Yaskawa INFORM job: DEMO_ROOF_SIDE_0625_3PAINT_43.JBI

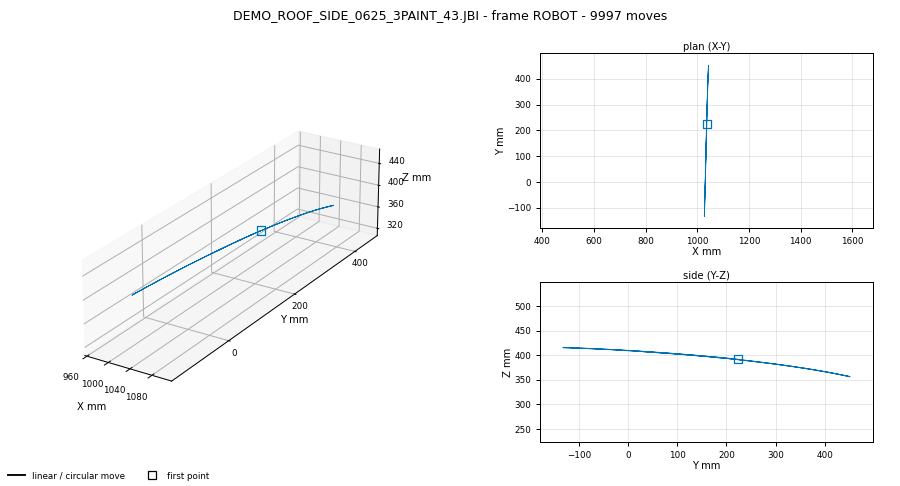
[picture p0: tool path of DEMO_ROOF_SIDE_0625_3PAINT_43.JBI in frame ROBOT, 9997 of 9997 moves have a stored position in this frame; points joined in program order, loops and branches not executed]
/JOB
//NAME DEMO_ROOF_SIDE_0625_3PAINT43
//POS
///NPOS 9997,0,0,0,0,0
///TOOL 0
///USER 0
///POSTYPE ROBOT
///RECTAN
///RCONF 1,0,0,0,0,0,0,0,0,0,0,0,0,0,0,0,0,0,0,0,0,0,0,0
C00000=1036.877,223.330,392.061,170.729,42.269,158.043
C00001=1036.870,223.081,392.088,170.727,42.268,158.043
C00002=1036.863,222.832,392.115,170.723,42.267,158.042
C00003=1036.857,222.584,392.143,170.721,42.266,158.042
C00004=1036.850,222.336,392.170,170.718,42.265,158.042
C00005=1036.844,222.088,392.198,170.716,42.264,158.041
C00006=1036.837,221.839,392.225,170.713,42.263,158.041
C00007=1036.830,221.591,392.252,170.711,42.262,158.040
C00008=1036.823,221.342,392.280,170.709,42.261,158.040
C00009=1036.817,221.094,392.307,170.705,42.261,158.040
C00010=1036.808,220.760,392.343,170.703,42.259,158.039
C00011=1036.799,220.427,392.380,170.699,42.258,158.039
C00012=1036.790,220.094,392.416,170.696,42.257,158.038
C00013=1036.782,219.761,392.454,170.692,42.255,158.038
C00014=1036.775,219.512,392.480,170.690,42.254,158.037
C00015=1036.768,219.264,392.508,170.687,42.254,158.037
C00016=1036.761,219.015,392.535,170.685,42.253,158.037
C00017=1036.754,218.767,392.562,170.683,42.252,158.036
C00018=1036.748,218.518,392.590,170.679,42.251,158.036
C00019=1036.741,218.270,392.616,170.677,42.251,158.036
C00020=1036.734,218.022,392.643,170.674,42.250,158.035
C00021=1036.727,217.773,392.670,170.672,42.249,158.035
C00022=1036.721,217.525,392.697,170.669,42.248,158.035
C00023=1036.714,217.276,392.724,170.667,42.247,158.034
C00024=1036.707,217.028,392.751,170.665,42.246,158.034
C00025=1036.701,216.779,392.778,170.662,42.245,158.034
C00026=1036.694,216.531,392.805,170.659,42.245,158.033
C00027=1036.687,216.282,392.832,170.657,42.244,158.033
C00028=1036.680,216.034,392.859,170.654,42.243,158.033
C00029=1036.674,215.785,392.886,170.652,42.242,158.032
C00030=1036.667,215.537,392.913,170.649,42.241,158.032
C00031=1036.660,215.288,392.940,170.647,42.240,158.031
C00032=1036.654,215.040,392.966,170.645,42.239,158.031
C00033=1036.647,214.792,392.994,170.642,42.238,158.031
C00034=1036.640,214.543,393.021,170.640,42.237,158.030
C00035=1036.634,214.295,393.048,170.637,42.236,158.030
C00036=1036.627,214.046,393.074,170.635,42.235,158.030
C00037=1036.620,213.797,393.101,170.633,42.234,158.029
C00038=1036.613,213.549,393.128,170.630,42.234,158.029
C00039=1036.607,213.301,393.155,170.628,42.233,158.029
C00040=1036.600,213.052,393.183,170.626,42.232,158.028
C00041=1036.593,212.804,393.209,170.622,42.231,158.028
C00042=1036.588,212.555,393.236,170.620,42.230,158.028
C00043=1036.580,212.307,393.263,170.617,42.229,158.027
C00044=1036.574,212.058,393.290,170.615,42.228,158.027
C00045=1036.567,211.810,393.316,170.612,42.227,158.027
C00046=1036.561,211.561,393.343,170.610,42.226,158.026
C00047=1036.553,211.313,393.370,170.608,42.226,158.026
C00048=1036.547,211.065,393.396,170.605,42.225,158.025
C00049=1036.541,210.816,393.423,170.603,42.224,158.025
C00050=1036.533,210.567,393.450,170.601,42.223,158.025
C00051=1036.527,210.319,393.477,170.598,42.222,158.025
C00052=1036.520,210.070,393.504,170.596,42.221,158.024
C00053=1036.513,209.822,393.530,170.593,42.220,158.024
C00054=1036.507,209.573,393.557,170.591,42.219,158.023
C00055=1036.500,209.325,393.583,170.589,42.219,158.023
C00056=1036.493,209.077,393.610,170.586,42.218,158.023
C00057=1036.487,208.828,393.637,170.584,42.217,158.022
C00058=1036.480,208.579,393.663,170.582,42.216,158.022
C00059=1036.473,208.331,393.689,170.579,42.215,158.022
C00060=1036.466,208.083,393.716,170.577,42.214,158.021
C00061=1036.460,207.834,393.743,170.574,42.213,158.021
C00062=1036.453,207.585,393.769,170.572,42.213,158.021
C00063=1036.446,207.337,393.795,170.570,42.212,158.020
C00064=1036.440,207.089,393.821,170.567,42.211,158.020
C00065=1036.433,206.840,393.848,170.565,42.210,158.020
C00066=1036.424,206.513,393.883,170.561,42.209,158.019
C00067=1036.415,206.185,393.919,170.559,42.208,158.019
C00068=1036.406,205.857,393.953,170.555,42.207,158.019
C00069=1036.398,205.530,393.988,170.552,42.206,158.018
C00070=1036.371,204.480,394.094,170.239,42.102,157.976
C00071=1036.365,204.230,394.118,170.236,42.101,157.976
C00072=1036.359,203.982,394.144,170.233,42.101,157.976
C00073=1036.353,203.733,394.169,170.230,42.101,157.975
C00074=1036.347,203.484,394.194,170.226,42.101,157.975
C00075=1036.340,203.236,394.220,170.223,42.101,157.975
C00076=1036.335,202.987,394.244,170.220,42.100,157.975
C00077=1036.329,202.739,394.269,170.217,42.100,157.974
C00078=1036.322,202.490,394.294,170.214,42.101,157.974
C00079=1036.316,202.241,394.319,170.211,42.100,157.974
C00080=1036.310,201.992,394.344,170.206,42.100,157.974
C00081=1036.304,201.744,394.369,170.203,42.100,157.973
C00082=1036.298,201.496,394.394,170.200,42.100,157.973
C00083=1036.292,201.246,394.419,170.197,42.100,157.973
C00084=1036.286,200.998,394.444,170.194,42.100,157.973
C00085=1036.280,200.749,394.470,170.190,42.100,157.973
C00086=1036.273,200.500,394.494,170.187,42.100,157.972
C00087=1036.267,200.251,394.519,170.184,42.100,157.972
C00088=1036.261,200.003,394.543,170.181,42.100,157.972
C00089=1036.255,199.754,394.568,170.178,42.100,157.972
C00090=1036.248,199.505,394.592,170.174,42.100,157.972
C00091=1036.242,199.257,394.617,170.171,42.100,157.971
C00092=1036.236,199.008,394.643,170.168,42.100,157.971
C00093=1036.230,198.760,394.666,170.165,42.100,157.971
C00094=1036.224,198.510,394.691,170.162,42.100,157.971
C00095=1036.217,198.262,394.716,170.159,42.100,157.971
C00096=1036.211,198.013,394.740,170.156,42.101,157.970
C00097=1036.204,197.764,394.765,170.152,42.100,157.970
C00098=1036.199,197.516,394.789,170.149,42.100,157.970
C00099=1036.192,197.268,394.814,170.146,42.101,157.970
C00100=1036.186,197.018,394.839,170.142,42.101,157.970
C00101=1036.179,196.770,394.863,170.139,42.100,157.969
C00102=1036.173,196.521,394.888,170.136,42.101,157.969
C00103=1036.167,196.272,394.912,170.132,42.101,157.969
C00104=1036.161,196.024,394.937,170.129,42.101,157.969
C00105=1036.155,195.774,394.962,170.126,42.101,157.969
C00106=1036.149,195.526,394.985,170.123,42.101,157.968
C00107=1036.142,195.277,395.011,170.120,42.101,157.968
C00108=1036.136,195.028,395.035,170.117,42.101,157.968
C00109=1036.131,194.780,395.059,170.114,42.101,157.968
C00110=1036.124,194.531,395.084,170.110,42.101,157.968
C00111=1036.118,194.282,395.108,170.107,42.102,157.968
C00112=1036.112,194.034,395.132,170.104,42.102,157.967
C00113=1036.105,193.785,395.157,170.101,42.101,157.967
C00114=1036.099,193.536,395.181,170.099,42.102,157.967
C00115=1036.093,193.288,395.206,170.096,42.101,157.967
C00116=1036.087,193.039,395.230,170.093,42.102,157.967
C00117=1036.081,192.790,395.255,170.089,42.102,157.966
C00118=1036.075,192.542,395.279,170.086,42.102,157.966
C00119=1036.069,192.292,395.303,170.083,42.102,157.966
C00120=1036.063,192.044,395.327,170.080,42.102,157.966
C00121=1036.057,191.795,395.352,170.077,42.102,157.966
C00122=1036.050,191.547,395.376,170.074,42.102,157.965
C00123=1036.045,191.298,395.401,170.071,42.102,157.965
C00124=1036.038,191.049,395.425,170.067,42.102,157.965
C00125=1036.033,190.800,395.449,170.064,42.103,157.965
C00126=1036.026,190.551,395.473,170.061,42.103,157.965
C00127=1036.020,190.302,395.497,170.058,42.103,157.965
C00128=1036.014,190.054,395.522,170.055,42.103,157.964
C00129=1036.008,189.805,395.546,170.052,42.103,157.964
C00130=1036.002,189.557,395.570,170.049,42.103,157.964
C00131=1035.995,189.272,395.597,170.046,42.103,157.964
C00132=1035.988,188.989,395.625,170.042,42.103,157.964
C00133=1035.981,188.704,395.653,170.038,42.104,157.964
C00134=1035.974,188.420,395.680,170.035,42.104,157.963
C00135=1035.968,188.171,395.705,170.032,42.103,157.963
C00136=1035.962,187.923,395.729,170.029,42.104,157.963
C00137=1035.956,187.673,395.753,170.026,42.104,157.963
C00138=1035.950,187.425,395.777,170.024,42.104,157.963
C00139=1035.944,187.176,395.801,170.020,42.104,157.962
C00140=1035.938,186.927,395.825,170.017,42.104,157.962
C00141=1035.932,186.678,395.850,170.014,42.105,157.962
C00142=1035.926,186.430,395.873,170.011,42.105,157.962
C00143=1035.921,186.181,395.898,170.008,42.105,157.962
C00144=1035.914,185.932,395.922,170.005,42.105,157.962
C00145=1035.909,185.684,395.946,170.002,42.105,157.961
C00146=1035.903,185.435,395.970,170.000,42.105,157.961
C00147=1035.896,185.186,395.994,169.997,42.105,157.961
C00148=1035.891,184.937,396.018,169.993,42.105,157.961
C00149=1035.885,184.689,396.042,169.990,42.106,157.961
C00150=1035.879,184.440,396.067,169.987,42.105,157.961
C00151=1035.873,184.191,396.090,169.984,42.106,157.960
C00152=1035.867,183.943,396.114,169.982,42.105,157.960
C00153=1035.861,183.693,396.138,169.979,42.106,157.960
C00154=1035.856,183.445,396.162,169.976,42.106,157.960
C00155=1035.849,183.196,396.186,169.972,42.106,157.960
C00156=1035.843,182.947,396.210,169.969,42.107,157.960
C00157=1035.837,182.698,396.233,169.966,42.107,157.960
C00158=1035.831,182.449,396.257,169.963,42.108,157.959
C00159=1035.823,182.201,396.280,169.960,42.108,157.959
C00160=1035.818,181.952,396.303,169.957,42.108,157.959
C00161=1035.811,181.703,396.327,169.955,42.108,157.959
C00162=1035.805,181.454,396.350,169.952,42.109,157.959
C00163=1035.799,181.205,396.374,169.949,42.109,157.959
C00164=1035.793,180.957,396.398,169.946,42.109,157.959
C00165=1035.787,180.708,396.421,169.943,42.110,157.959
C00166=1035.780,180.459,396.445,169.940,42.110,157.958
C00167=1035.774,180.210,396.468,169.937,42.110,157.958
C00168=1035.767,179.961,396.491,169.934,42.111,157.958
C00169=1035.761,179.712,396.514,169.931,42.111,157.958
C00170=1035.755,179.463,396.538,169.929,42.111,157.958
C00171=1035.749,179.215,396.562,169.926,42.112,157.958
C00172=1035.743,178.966,396.585,169.923,42.112,157.958
C00173=1035.736,178.717,396.609,169.919,42.113,157.958
C00174=1035.731,178.468,396.632,169.916,42.113,157.958
C00175=1035.723,178.220,396.655,169.913,42.114,157.957
C00176=1035.717,177.971,396.678,169.910,42.113,157.957
C00177=1035.712,177.722,396.701,169.908,42.114,157.957
C00178=1035.705,177.473,396.725,169.905,42.114,157.957
C00179=1035.699,177.224,396.748,169.902,42.115,157.957
C00180=1035.693,176.975,396.772,169.899,42.115,157.957
C00181=1035.687,176.726,396.795,169.896,42.115,157.957
C00182=1035.680,176.478,396.818,169.893,42.116,157.957
C00183=1035.674,176.229,396.841,169.891,42.116,157.957
C00184=1035.668,175.980,396.864,169.888,42.117,157.956
C00185=1035.662,175.731,396.888,169.885,42.117,157.956
C00186=1035.656,175.482,396.911,169.882,42.117,157.956
C00187=1035.650,175.234,396.935,169.879,42.117,157.956
C00188=1035.644,174.985,396.958,169.876,42.118,157.956
C00189=1035.637,174.736,396.980,169.874,42.118,157.956
C00190=1035.631,174.487,397.004,169.871,42.118,157.956
C00191=1035.625,174.238,397.027,169.867,42.119,157.956
C00192=1035.619,173.989,397.050,169.864,42.119,157.955
C00193=1035.613,173.740,397.074,169.861,42.120,157.955
C00194=1035.607,173.491,397.097,169.859,42.120,157.955
C00195=1035.600,173.207,397.123,169.855,42.121,157.955
C00196=1035.592,172.922,397.149,169.852,42.121,157.955
C00197=1035.586,172.638,397.176,169.849,42.122,157.955
C00198=1035.579,172.354,397.202,169.846,42.122,157.955
C00199=1035.573,172.104,397.225,169.843,42.122,157.955
C00200=1035.567,171.856,397.249,169.840,42.122,157.954
C00201=1035.561,171.607,397.272,169.838,42.123,157.954
C00202=1035.554,171.359,397.294,169.835,42.123,157.954
C00203=1035.548,171.109,397.318,169.832,42.123,157.954
C00204=1035.542,170.860,397.341,169.829,42.124,157.954
C00205=1035.536,170.612,397.364,169.827,42.124,157.954
C00206=1035.531,170.363,397.387,169.824,42.125,157.954
C00207=1035.525,170.114,397.410,169.821,42.125,157.954
C00208=1035.518,169.865,397.433,169.818,42.126,157.954
C00209=1035.512,169.616,397.456,169.816,42.126,157.954
C00210=1035.506,169.367,397.479,169.813,42.126,157.953
C00211=1035.500,169.119,397.503,169.810,42.127,157.953
C00212=1035.495,168.870,397.525,169.807,42.127,157.953
C00213=1035.488,168.621,397.548,169.804,42.127,157.953
C00214=1035.482,168.371,397.571,169.801,42.128,157.953
C00215=1035.476,168.123,397.594,169.798,42.128,157.953
C00216=1035.470,167.874,397.617,169.796,42.129,157.953
C00217=1035.465,167.625,397.640,169.793,42.129,157.953
C00218=1035.458,167.376,397.662,169.790,42.129,157.953
C00219=1035.452,167.127,397.685,169.787,42.129,157.952
C00220=1035.447,166.878,397.708,169.785,42.130,157.952
C00221=1035.441,166.630,397.732,169.782,42.130,157.952
C00222=1035.434,166.381,397.755,169.779,42.131,157.952
C00223=1035.428,166.132,397.778,169.777,42.131,157.952
C00224=1035.422,165.883,397.800,169.774,42.131,157.952
C00225=1035.416,165.634,397.823,169.771,42.132,157.952
C00226=1035.411,165.385,397.846,169.769,42.132,157.952
C00227=1035.404,165.137,397.869,169.766,42.132,157.952
C00228=1035.398,164.888,397.892,169.763,42.133,157.952
C00229=1035.393,164.639,397.915,169.761,42.133,157.951
C00230=1035.387,164.390,397.938,169.758,42.134,157.951
C00231=1035.381,164.141,397.960,169.755,42.134,157.951
C00232=1035.375,163.893,397.983,169.753,42.134,157.951
C00233=1035.369,163.643,398.005,169.750,42.135,157.951
C00234=1035.364,163.394,398.028,169.747,42.135,157.951
C00235=1035.358,163.145,398.051,169.745,42.136,157.951
C00236=1035.351,162.897,398.073,169.742,42.136,157.951
C00237=1035.346,162.648,398.096,169.738,42.136,157.951
C00238=1035.340,162.399,398.119,169.736,42.137,157.951
C00239=1035.334,162.150,398.142,169.733,42.137,157.951
C00240=1035.328,161.901,398.164,169.730,42.138,157.950
C00241=1035.322,161.652,398.187,169.728,42.138,157.950
C00242=1035.316,161.404,398.210,169.725,42.138,157.950
C00243=1035.311,161.154,398.233,169.722,42.139,157.950
C00244=1035.304,160.905,398.255,169.720,42.139,157.950
C00245=1035.299,160.657,398.278,169.717,42.140,157.950
C00246=1035.293,160.408,398.301,169.715,42.140,157.950
C00247=1035.287,160.159,398.324,169.712,42.140,157.950
C00248=1035.282,159.909,398.346,169.709,42.141,157.950
C00249=1035.275,159.661,398.368,169.707,42.141,157.950
C00250=1035.269,159.412,398.391,169.704,42.141,157.949
C00251=1035.263,159.163,398.414,169.701,42.142,157.949
C00252=1035.257,158.914,398.435,169.699,42.142,157.949
C00253=1035.250,158.665,398.458,169.696,42.143,157.949
C00254=1035.245,158.416,398.480,169.693,42.144,157.949
C00255=1035.238,158.167,398.503,169.691,42.144,157.949
C00256=1035.232,157.918,398.525,169.688,42.145,157.949
C00257=1035.226,157.668,398.547,169.685,42.145,157.949
C00258=1035.220,157.421,398.569,169.683,42.146,157.949
C00259=1035.213,157.135,398.595,169.679,42.146,157.949
C00260=1035.206,156.850,398.620,169.676,42.147,157.949
C00261=1035.199,156.565,398.646,169.673,42.147,157.949
C00262=1035.192,156.280,398.671,169.670,42.148,157.949
C00263=1035.186,156.032,398.694,169.668,42.149,157.949
C00264=1035.180,155.782,398.716,169.665,42.149,157.948
C00265=1035.174,155.533,398.738,169.662,42.150,157.948
C00266=1035.168,155.284,398.760,169.660,42.150,157.948
C00267=1035.162,155.035,398.783,169.657,42.151,157.948
C00268=1035.156,154.786,398.804,169.655,42.151,157.948
C00269=1035.150,154.538,398.826,169.652,42.152,157.948
C00270=1035.144,154.289,398.848,169.649,42.152,157.948
C00271=1035.138,154.040,398.871,169.647,42.153,157.948
C00272=1035.132,153.791,398.893,169.644,42.154,157.948
C00273=1035.125,153.542,398.915,169.641,42.154,157.948
C00274=1035.119,153.293,398.937,169.639,42.154,157.948
C00275=1035.114,153.044,398.959,169.636,42.155,157.948
C00276=1035.107,152.795,398.981,169.633,42.156,157.948
C00277=1035.101,152.546,399.003,169.631,42.156,157.948
C00278=1035.095,152.297,399.025,169.628,42.157,157.948
C00279=1035.088,152.048,399.047,169.626,42.158,157.948
C00280=1035.082,151.799,399.068,169.623,42.158,157.947
C00281=1035.077,151.551,399.091,169.620,42.158,157.947
C00282=1035.071,151.301,399.113,169.618,42.159,157.947
C00283=1035.065,151.052,399.134,169.615,42.160,157.947
C00284=1035.058,150.804,399.157,169.613,42.160,157.947
C00285=1035.052,150.554,399.178,169.610,42.161,157.947
C00286=1035.046,150.305,399.200,169.607,42.162,157.947
C00287=1035.040,150.056,399.223,169.605,42.162,157.947
C00288=1035.034,149.807,399.244,169.602,42.162,157.947
C00289=1035.029,149.559,399.266,169.601,42.163,157.947
C00290=1035.022,149.310,399.288,169.598,42.164,157.947
C00291=1035.016,149.061,399.310,169.594,42.164,157.947
C00292=1035.010,148.812,399.331,169.593,42.165,157.947
C00293=1035.004,148.562,399.353,169.590,42.166,157.947
C00294=1034.998,148.314,399.376,169.588,42.166,157.947
C00295=1034.992,148.065,399.397,169.585,42.166,157.947
C00296=1034.986,147.816,399.419,169.582,42.167,157.947
C00297=1034.980,147.567,399.440,169.580,42.168,157.947
C00298=1034.974,147.318,399.463,169.577,42.168,157.946
C00299=1034.967,147.069,399.484,169.575,42.169,157.947
C00300=1034.961,146.820,399.506,169.572,42.170,157.946
C00301=1034.956,146.571,399.527,169.569,42.171,157.946
C00302=1034.949,146.322,399.549,169.567,42.171,157.946
C00303=1034.943,146.073,399.571,169.564,42.171,157.946
C00304=1034.937,145.823,399.592,169.562,42.172,157.946
C00305=1034.931,145.574,399.614,169.559,42.173,157.946
C00306=1034.925,145.326,399.636,169.556,42.174,157.946
C00307=1034.918,145.078,399.657,169.554,42.174,157.946
C00308=1034.912,144.828,399.679,169.551,42.175,157.946
C00309=1034.906,144.579,399.700,169.549,42.176,157.946
C00310=1034.900,144.330,399.722,169.546,42.176,157.946
C00311=1034.894,144.081,399.743,169.544,42.177,157.946
C00312=1034.888,143.832,399.765,169.541,42.177,157.946
C00313=1034.882,143.583,399.786,169.538,42.178,157.946
C00314=1034.876,143.334,399.808,169.536,42.179,157.946
C00315=1034.870,143.085,399.830,169.533,42.179,157.946
C00316=1034.864,142.836,399.851,169.532,42.180,157.946
C00317=1034.857,142.587,399.872,169.528,42.181,157.946
C00318=1034.851,142.338,399.894,169.527,42.182,157.946
C00319=1034.845,142.089,399.915,169.524,42.182,157.946
C00320=1034.839,141.840,399.936,169.521,42.183,157.946
C00321=1034.833,141.591,399.958,169.519,42.183,157.946
C00322=1034.827,141.342,399.980,169.516,42.184,157.946
C00323=1034.821,141.056,400.004,169.513,42.185,157.946
C00324=1034.813,140.771,400.028,169.511,42.185,157.946
C00325=1034.807,140.486,400.053,169.508,42.186,157.946
C00326=1034.799,140.200,400.077,169.505,42.187,157.945
C00327=1034.794,139.952,400.099,169.502,42.187,157.945
C00328=1034.787,139.702,400.120,169.500,42.188,157.945
C00329=1034.781,139.453,400.142,169.497,42.189,157.945
C00330=1034.776,139.205,400.163,169.495,42.190,157.945
C00331=1034.769,138.956,400.184,169.492,42.190,157.945
C00332=1034.763,138.707,400.206,169.490,42.191,157.945
C00333=1034.756,138.457,400.227,169.487,42.191,157.945
C00334=1034.751,138.208,400.248,169.484,42.193,157.945
C00335=1034.744,137.959,400.269,169.482,42.193,157.945
C00336=1034.738,137.710,400.291,169.479,42.193,157.945
C00337=1034.733,137.462,400.312,169.477,42.194,157.945
C00338=1034.726,137.213,400.333,169.474,42.195,157.945
C00339=1034.720,136.963,400.354,169.473,42.196,157.945
C00340=1034.714,136.715,400.375,169.470,42.196,157.945
C00341=1034.708,136.465,400.397,169.468,42.197,157.945
C00342=1034.701,136.216,400.418,169.465,42.197,157.945
C00343=1034.696,135.967,400.438,169.463,42.198,157.945
C00344=1034.690,135.718,400.460,169.460,42.199,157.945
C00345=1034.683,135.469,400.481,169.458,42.200,157.945
C00346=1034.678,135.220,400.502,169.455,42.201,157.945
C00347=1034.671,134.971,400.523,169.452,42.201,157.945
C00348=1034.664,134.722,400.544,169.450,42.202,157.945
C00349=1034.659,134.473,400.565,169.447,42.203,157.945
C00350=1034.652,134.224,400.586,169.445,42.204,157.945
C00351=1034.647,133.975,400.607,169.442,42.204,157.945
C00352=1034.641,133.726,400.628,169.440,42.205,157.945
C00353=1034.634,133.477,400.649,169.437,42.206,157.945
C00354=1034.628,133.228,400.670,169.436,42.206,157.945
C00355=1034.622,132.979,400.691,169.433,42.207,157.945
C00356=1034.616,132.730,400.712,169.431,42.208,157.945
C00357=1034.610,132.481,400.734,169.428,42.208,157.945
C00358=1034.604,132.231,400.754,169.426,42.209,157.945
C00359=1034.598,131.983,400.775,169.423,42.210,157.945
C00360=1034.592,131.733,400.796,169.421,42.211,157.945
C00361=1034.586,131.485,400.817,169.418,42.211,157.944
C00362=1034.580,131.235,400.838,169.416,42.212,157.945
C00363=1034.573,130.986,400.859,169.413,42.212,157.944
C00364=1034.568,130.737,400.879,169.411,42.213,157.945
C00365=1034.561,130.488,400.900,169.408,42.214,157.944
C00366=1034.556,130.239,400.921,169.406,42.215,157.944
C00367=1034.549,129.990,400.942,169.403,42.216,157.944
C00368=1034.542,129.741,400.962,169.401,42.216,157.944
C00369=1034.537,129.492,400.984,169.399,42.217,157.944
C00370=1034.530,129.243,401.004,169.397,42.218,157.945
C00371=1034.524,128.994,401.025,169.394,42.219,157.944
C00372=1034.517,128.745,401.045,169.392,42.220,157.944
C00373=1034.511,128.495,401.066,169.389,42.221,157.944
C00374=1034.505,128.247,401.087,169.387,42.221,157.944
C00375=1034.498,127.997,401.107,169.384,42.222,157.944
C00376=1034.493,127.748,401.127,169.382,42.223,157.944
C00377=1034.486,127.499,401.148,169.379,42.224,157.944
C00378=1034.480,127.251,401.168,169.376,42.225,157.944
C00379=1034.474,127.001,401.190,169.375,42.226,157.944
C00380=1034.468,126.753,401.210,169.371,42.226,157.944
C00381=1034.461,126.503,401.230,169.370,42.227,157.944
C00382=1034.455,126.254,401.251,169.367,42.228,157.944
C00383=1034.449,126.005,401.272,169.365,42.228,157.944
C00384=1034.443,125.756,401.292,169.362,42.229,157.944
C00385=1034.437,125.507,401.312,169.360,42.230,157.944
C00386=1034.431,125.258,401.334,169.357,42.231,157.944
C00387=1034.423,124.972,401.357,169.355,42.232,157.944
C00388=1034.416,124.687,401.381,169.352,42.233,157.944
C00389=1034.409,124.401,401.403,169.350,42.234,157.944
C00390=1034.402,124.116,401.427,169.346,42.234,157.944
C00391=1034.396,123.867,401.448,169.345,42.235,157.944
C00392=1034.390,123.618,401.469,169.342,42.237,157.944
C00393=1034.384,123.369,401.489,169.340,42.237,157.944
C00394=1034.377,123.119,401.509,169.337,42.238,157.944
C00395=1034.371,122.870,401.529,169.335,42.238,157.944
C00396=1034.365,122.621,401.551,169.332,42.239,157.944
C00397=1034.359,122.372,401.571,169.330,42.240,157.944
C00398=1034.353,122.124,401.591,169.327,42.241,157.944
C00399=1034.347,121.874,401.611,169.325,42.242,157.944
C00400=1034.341,121.625,401.631,169.322,42.243,157.944
C00401=1034.334,121.376,401.652,169.320,42.243,157.944
C00402=1034.328,121.127,401.672,169.318,42.244,157.944
C00403=1034.323,120.877,401.693,169.316,42.245,157.944
C00404=1034.317,120.629,401.713,169.314,42.245,157.944
C00405=1034.311,120.380,401.733,169.311,42.246,157.944
C00406=1034.304,120.130,401.754,169.309,42.247,157.944
C00407=1034.298,119.882,401.775,169.306,42.248,157.944
C00408=1034.292,119.632,401.795,169.304,42.249,157.944
C00409=1034.286,119.384,401.815,169.301,42.249,157.944
C00410=1034.280,119.135,401.835,169.299,42.250,157.944
C00411=1034.274,118.885,401.856,169.296,42.251,157.944
C00412=1034.268,118.636,401.876,169.294,42.252,157.944
C00413=1034.261,118.387,401.896,169.293,42.253,157.944
C00414=1034.255,118.138,401.916,169.289,42.253,157.944
C00415=1034.250,117.889,401.937,169.288,42.254,157.944
C00416=1034.244,117.639,401.957,169.285,42.255,157.944
C00417=1034.237,117.391,401.978,169.283,42.255,157.944
C00418=1034.231,117.142,401.998,169.280,42.256,157.944
C00419=1034.225,116.892,402.019,169.278,42.257,157.944
C00420=1034.219,116.643,402.039,169.276,42.258,157.944
C00421=1034.213,116.395,402.059,169.273,42.259,157.944
C00422=1034.207,116.145,402.079,169.271,42.259,157.944
C00423=1034.202,115.896,402.099,169.268,42.260,157.944
C00424=1034.196,115.647,402.119,169.266,42.261,157.944
C00425=1034.189,115.398,402.140,169.263,42.262,157.944
C00426=1034.183,115.149,402.160,169.261,42.262,157.944
C00427=1034.177,114.900,402.180,169.260,42.263,157.944
C00428=1034.171,114.650,402.201,169.257,42.264,157.944
C00429=1034.165,114.401,402.221,169.255,42.264,157.944
C00430=1034.159,114.153,402.241,169.252,42.265,157.944
C00431=1034.153,113.903,402.261,169.250,42.266,157.944
C00432=1034.148,113.653,402.281,169.248,42.267,157.944
C00433=1034.142,113.405,402.301,169.245,42.268,157.944
C00434=1034.135,113.155,402.321,169.243,42.268,157.944
C00435=1034.129,112.906,402.341,169.240,42.269,157.944
C00436=1034.123,112.657,402.361,169.238,42.270,157.944
C00437=1034.116,112.408,402.381,169.236,42.270,157.944
C00438=1034.110,112.159,402.401,169.233,42.271,157.944
C00439=1034.105,111.910,402.420,169.232,42.272,157.944
C00440=1034.099,111.661,402.440,169.229,42.274,157.944
C00441=1034.092,111.411,402.461,169.227,42.274,157.944
C00442=1034.086,111.162,402.481,169.224,42.275,157.944
C00443=1034.080,110.914,402.501,169.222,42.276,157.944
C00444=1034.074,110.664,402.520,169.220,42.276,157.944
C00445=1034.068,110.415,402.540,169.217,42.277,157.944
C00446=1034.061,110.166,402.560,169.215,42.278,157.944
C00447=1034.055,109.917,402.580,169.213,42.279,157.944
C00448=1034.049,109.667,402.599,169.210,42.280,157.944
C00449=1034.043,109.418,402.619,169.208,42.281,157.944
C00450=1034.037,109.170,402.639,169.206,42.282,157.944
C00451=1034.029,108.884,402.661,169.203,42.283,157.944
C00452=1034.022,108.598,402.684,169.200,42.284,157.944
C00453=1034.015,108.312,402.707,169.198,42.285,157.944
C00454=1034.008,108.027,402.729,169.195,42.286,157.944
C00455=1034.002,107.778,402.749,169.192,42.286,157.944
C00456=1033.996,107.529,402.769,169.190,42.287,157.944
C00457=1033.989,107.279,402.788,169.188,42.288,157.944
C00458=1033.983,107.030,402.808,169.186,42.289,157.944
C00459=1033.977,106.781,402.827,169.184,42.290,157.944
C00460=1033.971,106.532,402.847,169.181,42.291,157.944
C00461=1033.965,106.282,402.867,169.179,42.292,157.944
C00462=1033.958,106.033,402.886,169.176,42.293,157.944
C00463=1033.952,105.785,402.906,169.174,42.294,157.944
C00464=1033.946,105.536,402.926,169.171,42.294,157.944
C00465=1033.940,105.286,402.945,169.170,42.295,157.944
C00466=1033.933,105.037,402.965,169.168,42.296,157.944
C00467=1033.927,104.788,402.984,169.165,42.297,157.944
C00468=1033.921,104.539,403.004,169.163,42.298,157.944
C00469=1033.916,104.289,403.023,169.160,42.299,157.944
C00470=1033.910,104.041,403.043,169.158,42.300,157.944
C00471=1033.903,103.791,403.062,169.156,42.301,157.945
C00472=1033.897,103.542,403.082,169.153,42.301,157.944
C00473=1033.891,103.293,403.102,169.151,42.302,157.944
C00474=1033.885,103.044,403.122,169.149,42.303,157.945
C00475=1033.878,102.795,403.141,169.147,42.304,157.945
C00476=1033.873,102.546,403.160,169.145,42.304,157.944
C00477=1033.866,102.296,403.180,169.142,42.305,157.945
C00478=1033.860,102.047,403.200,169.140,42.306,157.945
C00479=1033.854,101.798,403.219,169.137,42.308,157.945
C00480=1033.848,101.549,403.238,169.135,42.308,157.945
C00481=1033.842,101.299,403.258,169.133,42.309,157.945
C00482=1033.836,101.051,403.278,169.130,42.310,157.945
C00483=1033.829,100.801,403.297,169.129,42.311,157.945
C00484=1033.823,100.552,403.316,169.127,42.311,157.945
C00485=1033.818,100.303,403.336,169.124,42.312,157.945
C00486=1033.812,100.054,403.356,169.122,42.313,157.945
C00487=1033.805,99.805,403.374,169.119,42.314,157.945
C00488=1033.799,99.555,403.394,169.117,42.315,157.945
C00489=1033.792,99.306,403.413,169.114,42.316,157.945
C00490=1033.786,99.057,403.433,169.112,42.317,157.945
C00491=1033.780,98.807,403.451,169.110,42.318,157.945
C00492=1033.774,98.559,403.471,169.108,42.319,157.945
C00493=1033.768,98.310,403.490,169.106,42.320,157.945
C00494=1033.762,98.060,403.509,169.103,42.321,157.945
C00495=1033.755,97.811,403.528,169.101,42.321,157.945
C00496=1033.749,97.562,403.548,169.099,42.322,157.945
C00497=1033.742,97.312,403.567,169.096,42.323,157.945
C00498=1033.737,97.063,403.586,169.094,42.324,157.945
C00499=1033.730,96.814,403.605,169.091,42.325,157.945
C00500=1033.724,96.565,403.625,169.090,42.326,157.945
C00501=1033.718,96.316,403.643,169.088,42.327,157.945
C00502=1033.712,96.066,403.662,169.085,42.328,157.945
C00503=1033.706,95.818,403.682,169.083,42.329,157.945
C00504=1033.699,95.569,403.700,169.080,42.330,157.945
C00505=1033.693,95.319,403.720,169.078,42.331,157.945
C00506=1033.687,95.070,403.738,169.076,42.332,157.945
C00507=1033.681,94.820,403.758,169.073,42.333,157.945
C00508=1033.674,94.572,403.777,169.071,42.333,157.945
C00509=1033.668,94.322,403.797,169.069,42.334,157.945
C00510=1033.662,94.073,403.815,169.067,42.335,157.945
C00511=1033.656,93.824,403.834,169.065,42.336,157.945
C00512=1033.650,93.574,403.853,169.062,42.337,157.945
C00513=1033.644,93.325,403.872,169.060,42.337,157.945
C00514=1033.637,93.077,403.892,169.057,42.338,157.945
C00515=1033.631,92.791,403.913,169.055,42.339,157.945
C00516=1033.623,92.505,403.935,169.053,42.341,157.945
C00517=1033.616,92.219,403.957,169.050,42.342,157.945
C00518=1033.609,91.934,403.979,169.047,42.343,157.945
C00519=1033.603,91.685,403.998,169.045,42.344,157.945
C00520=1033.597,91.435,404.017,169.043,42.345,157.945
C00521=1033.591,91.186,404.035,169.040,42.345,157.945
C00522=1033.585,90.937,404.055,169.038,42.346,157.945
C00523=1033.579,90.688,404.073,169.036,42.347,157.945
C00524=1033.573,90.438,404.093,169.034,42.348,157.945
C00525=1033.567,90.189,404.111,169.032,42.349,157.946
C00526=1033.561,89.940,404.130,169.029,42.350,157.945
C00527=1033.554,89.691,404.149,169.027,42.351,157.945
C00528=1033.548,89.441,404.168,169.025,42.351,157.946
C00529=1033.542,89.192,404.186,169.022,42.353,157.946
C00530=1033.535,88.943,404.205,169.020,42.354,157.946
C00531=1033.530,88.694,404.224,169.017,42.355,157.946
C00532=1033.523,88.445,404.243,169.016,42.356,157.946
C00533=1033.517,88.196,404.262,169.014,42.357,157.946
C00534=1033.510,87.946,404.280,169.011,42.358,157.946
C00535=1033.504,87.697,404.299,169.009,42.359,157.946
C00536=1033.497,87.448,404.318,169.006,42.360,157.946
C00537=1033.492,87.199,404.337,169.004,42.361,157.946
C00538=1033.485,86.950,404.355,169.002,42.361,157.946
C00539=1033.479,86.701,404.374,168.999,42.362,157.946
C00540=1033.472,86.451,404.393,168.998,42.363,157.946
C00541=1033.466,86.202,404.411,168.995,42.364,157.946
C00542=1033.460,85.953,404.429,168.993,42.365,157.946
C00543=1033.454,85.703,404.449,168.991,42.366,157.946
C00544=1033.448,85.454,404.467,168.988,42.367,157.946
C00545=1033.441,85.205,404.486,168.986,42.368,157.946
C00546=1033.435,84.956,404.505,168.984,42.369,157.946
C00547=1033.428,84.707,404.523,168.982,42.370,157.946
C00548=1033.422,84.457,404.541,168.980,42.371,157.946
C00549=1033.417,84.207,404.560,168.977,42.372,157.946
C00550=1033.410,83.958,404.579,168.975,42.373,157.946
C00551=1033.404,83.709,404.598,168.972,42.374,157.946
C00552=1033.398,83.461,404.616,168.970,42.375,157.946
C00553=1033.392,83.212,404.635,168.968,42.376,157.946
C00554=1033.385,82.962,404.653,168.966,42.377,157.946
C00555=1033.379,82.713,404.671,168.964,42.378,157.946
C00556=1033.373,82.463,404.690,168.961,42.379,157.946
C00557=1033.367,82.214,404.709,168.959,42.379,157.946
C00558=1033.361,81.964,404.727,168.957,42.380,157.946
C00559=1033.354,81.715,404.746,168.954,42.381,157.946
C00560=1033.348,81.466,404.764,168.952,42.382,157.946
C00561=1033.342,81.217,404.783,168.951,42.383,157.947
C00562=1033.336,80.968,404.800,168.948,42.384,157.947
C00563=1033.330,80.719,404.820,168.946,42.385,157.947
C00564=1033.324,80.470,404.838,168.943,42.386,157.947
C00565=1033.317,80.220,404.857,168.941,42.387,157.947
C00566=1033.311,79.971,404.875,168.939,42.388,157.947
C00567=1033.305,79.722,404.894,168.936,42.389,157.947
C00568=1033.298,79.472,404.912,168.934,42.390,157.947
C00569=1033.293,79.223,404.930,168.933,42.391,157.947
C00570=1033.287,78.974,404.949,168.930,42.392,157.947
C00571=1033.281,78.725,404.968,168.928,42.392,157.947
C00572=1033.275,78.475,404.986,168.926,42.393,157.947
C00573=1033.268,78.226,405.004,168.923,42.394,157.947
C00574=1033.262,77.977,405.023,168.921,42.395,157.947
C00575=1033.256,77.728,405.041,168.918,42.396,157.947
C00576=1033.250,77.479,405.059,168.916,42.397,157.947
C00577=1033.244,77.229,405.077,168.915,42.398,157.947
C00578=1033.237,76.980,405.096,168.912,42.399,157.947
C00579=1033.230,76.695,405.116,168.909,42.400,157.947
C00580=1033.223,76.408,405.138,168.907,42.401,157.947
C00581=1033.216,76.123,405.159,168.904,42.402,157.947
C00582=1033.209,75.837,405.179,168.901,42.403,157.947
C00583=1033.202,75.588,405.197,168.900,42.404,157.947
C00584=1033.196,75.338,405.215,168.897,42.406,157.947
C00585=1033.190,75.089,405.234,168.895,42.407,157.947
C00586=1033.184,74.840,405.251,168.893,42.407,157.947
C00587=1033.177,74.591,405.270,168.890,42.409,157.947
C00588=1033.171,74.341,405.287,168.888,42.410,157.947
C00589=1033.165,74.092,405.306,168.885,42.411,157.947
C00590=1033.158,73.842,405.324,168.884,42.412,157.947
C00591=1033.153,73.594,405.342,168.882,42.413,157.947
C00592=1033.146,73.344,405.360,168.879,42.414,157.947
C00593=1033.140,73.095,405.379,168.877,42.414,157.947
C00594=1033.133,72.846,405.396,168.874,42.415,157.947
C00595=1033.127,72.597,405.415,168.872,42.416,157.947
C00596=1033.121,72.348,405.432,168.870,42.417,157.948
C00597=1033.115,72.098,405.450,168.867,42.418,157.948
C00598=1033.109,71.849,405.469,168.866,42.419,157.948
C00599=1033.103,71.599,405.487,168.864,42.420,157.948
C00600=1033.097,71.351,405.505,168.861,42.421,157.948
C00601=1033.090,71.101,405.523,168.859,42.422,157.948
C00602=1033.084,70.851,405.541,168.856,42.423,157.948
C00603=1033.077,70.602,405.559,168.854,42.424,157.948
C00604=1033.072,70.353,405.577,168.853,42.425,157.948
C00605=1033.066,70.104,405.595,168.850,42.426,157.948
C00606=1033.059,69.855,405.613,168.848,42.427,157.948
C00607=1033.052,69.605,405.631,168.845,42.428,157.948
C00608=1033.047,69.356,405.648,168.843,42.429,157.948
C00609=1033.040,69.107,405.667,168.841,42.430,157.948
C00610=1033.034,68.857,405.685,168.838,42.431,157.948
C00611=1033.028,68.608,405.702,168.836,42.432,157.948
C00612=1033.022,68.359,405.720,168.834,42.433,157.948
C00613=1033.016,68.109,405.738,168.832,42.434,157.948
C00614=1033.009,67.860,405.756,168.830,42.435,157.948
C00615=1033.003,67.611,405.773,168.827,42.436,157.948
C00616=1032.997,67.361,405.791,168.825,42.437,157.948
C00617=1032.990,67.112,405.809,168.822,42.438,157.948
C00618=1032.984,66.863,405.827,168.821,42.439,157.948
C00619=1032.978,66.614,405.845,168.819,42.440,157.948
C00620=1032.971,66.364,405.862,168.816,42.441,157.948
C00621=1032.966,66.116,405.880,168.814,42.442,157.948
C00622=1032.959,65.866,405.898,168.811,42.443,157.948
C00623=1032.953,65.617,405.916,168.809,42.444,157.948
C00624=1032.946,65.367,405.934,168.807,42.445,157.949
C00625=1032.940,65.118,405.951,168.805,42.446,157.949
C00626=1032.934,64.868,405.968,168.803,42.447,157.949
C00627=1032.928,64.619,405.987,168.800,42.448,157.949
C00628=1032.921,64.371,406.004,168.798,42.449,157.949
C00629=1032.915,64.121,406.022,168.796,42.450,157.949
C00630=1032.908,63.871,406.039,168.793,42.451,157.949
C00631=1032.903,63.622,406.057,168.792,42.452,157.949
C00632=1032.896,63.373,406.074,168.789,42.453,157.949
C00633=1032.890,63.123,406.092,168.787,42.454,157.949
C00634=1032.884,62.874,406.109,168.785,42.455,157.949
C00635=1032.877,62.625,406.127,168.782,42.456,157.949
C00636=1032.871,62.375,406.144,168.780,42.457,157.949
C00637=1032.864,62.127,406.161,168.777,42.458,157.949
C00638=1032.858,61.877,406.179,168.776,42.460,157.949
C00639=1032.851,61.627,406.197,168.773,42.461,157.949
C00640=1032.845,61.379,406.214,168.771,42.462,157.949
C00641=1032.838,61.129,406.231,168.768,42.463,157.949
C00642=1032.832,60.879,406.249,168.766,42.464,157.949
C00643=1032.823,60.524,406.273,168.763,42.466,157.949
C00644=1032.814,60.168,406.299,168.760,42.467,157.949
C00645=1032.805,59.812,406.323,168.756,42.469,157.950
C00646=1032.796,59.456,406.348,168.753,42.470,157.950
C00647=1032.790,59.207,406.365,168.752,42.471,157.950
C00648=1032.783,58.958,406.383,168.749,42.472,157.950
C00649=1032.776,58.709,406.400,168.747,42.473,157.950
C00650=1032.770,58.460,406.417,168.744,42.475,157.950
C00651=1032.765,58.245,406.432,168.742,42.476,157.950
C00652=1032.759,58.030,406.446,168.740,42.476,157.950
C00653=1032.754,57.816,406.462,168.738,42.477,157.950
C00654=1032.748,57.602,406.476,168.737,42.478,157.950
C00655=1032.743,57.387,406.492,168.735,42.479,157.950
C00656=1032.738,57.173,406.506,168.733,42.480,157.950
C00657=1032.733,56.959,406.521,168.731,42.481,157.950
C00658=1032.726,56.744,406.536,168.728,42.482,157.950
C00659=1032.721,56.495,406.553,168.726,42.483,157.950
C00660=1032.714,56.246,406.571,168.725,42.484,157.950
C00661=1032.708,55.997,406.588,168.722,42.485,157.950
C00662=1032.702,55.747,406.605,168.720,42.486,157.950
C00663=1032.696,55.498,406.622,168.717,42.488,157.950
C00664=1032.689,55.248,406.639,168.715,42.489,157.950
C00665=1032.683,54.999,406.657,168.712,42.490,157.950
C00666=1032.676,54.750,406.674,168.710,42.491,157.950
C00667=1032.670,54.500,406.691,168.709,42.492,157.951
C00668=1032.664,54.251,406.708,168.706,42.493,157.951
C00669=1032.657,54.001,406.726,168.704,42.494,157.951
C00670=1032.651,53.753,406.743,168.701,42.495,157.951
C00671=1032.645,53.503,406.759,168.699,42.496,157.951
C00672=1032.639,53.254,406.777,168.696,42.497,157.951
C00673=1032.632,53.004,406.794,168.695,42.498,157.951
C00674=1032.626,52.755,406.811,168.693,42.499,157.951
C00675=1032.620,52.505,406.828,168.690,42.501,157.951
C00676=1032.614,52.256,406.845,168.688,42.502,157.951
C00677=1032.607,52.007,406.863,168.685,42.503,157.951
C00678=1032.601,51.758,406.880,168.684,42.504,157.951
C00679=1032.595,51.508,406.897,168.682,42.505,157.951
C00680=1032.589,51.259,406.914,168.679,42.506,157.951
C00681=1032.582,51.010,406.931,168.677,42.507,157.951
C00682=1032.577,50.760,406.948,168.674,42.508,157.951
C00683=1032.570,50.511,406.965,168.672,42.509,157.951
C00684=1032.564,50.262,406.982,168.669,42.510,157.951
C00685=1032.558,50.013,406.999,168.667,42.510,157.951
C00686=1032.551,49.763,407.017,168.666,42.511,157.951
C00687=1032.545,49.514,407.033,168.663,42.512,157.951
C00688=1032.539,49.264,407.050,168.661,42.513,157.951
C00689=1032.532,49.015,407.067,168.658,42.514,157.951
C00690=1032.527,48.766,407.085,168.656,42.515,157.951
C00691=1032.520,48.516,407.101,168.654,42.516,157.951
C00692=1032.514,48.267,407.118,168.651,42.517,157.951
C00693=1032.508,48.017,407.135,168.650,42.518,157.951
C00694=1032.502,47.768,407.152,168.647,42.520,157.951
C00695=1032.496,47.520,407.169,168.645,42.521,157.952
C00696=1032.489,47.270,407.186,168.643,42.522,157.952
C00697=1032.484,47.021,407.204,168.640,42.523,157.952
C00698=1032.477,46.771,407.220,168.638,42.524,157.952
C00699=1032.471,46.522,407.237,168.636,42.525,157.952
C00700=1032.465,46.272,407.253,168.634,42.526,157.952
C00701=1032.459,46.023,407.271,168.632,42.527,157.952
C00702=1032.453,45.774,407.288,168.629,42.528,157.952
C00703=1032.446,45.524,407.305,168.627,42.529,157.952
C00704=1032.440,45.275,407.322,168.624,42.530,157.952
C00705=1032.434,45.026,407.339,168.623,42.531,157.952
C00706=1032.428,44.776,407.356,168.619,42.531,157.952
C00707=1032.421,44.490,407.375,168.618,42.533,157.952
C00708=1032.413,44.204,407.395,168.615,42.534,157.952
C00709=1032.407,43.917,407.414,168.612,42.535,157.952
C00710=1032.400,43.631,407.433,168.609,42.536,157.952
C00711=1032.394,43.382,407.450,168.607,42.537,157.952
C00712=1032.388,43.133,407.466,168.605,42.538,157.952
C00713=1032.381,42.883,407.484,168.603,42.539,157.952
C00714=1032.375,42.634,407.500,168.601,42.540,157.952
C00715=1032.369,42.385,407.516,168.598,42.541,157.952
C00716=1032.362,42.135,407.534,168.596,42.542,157.952
C00717=1032.356,41.886,407.550,168.593,42.544,157.952
C00718=1032.349,41.636,407.567,168.591,42.545,157.952
C00719=1032.343,41.387,407.583,168.590,42.546,157.952
C00720=1032.337,41.138,407.600,168.587,42.547,157.952
C00721=1032.331,40.888,407.617,168.585,42.548,157.952
C00722=1032.325,40.639,407.633,168.582,42.549,157.952
C00723=1032.319,40.390,407.650,168.580,42.550,157.952
C00724=1032.312,40.141,407.667,168.577,42.551,157.953
C00725=1032.306,39.891,407.683,168.576,42.552,157.953
C00726=1032.300,39.641,407.699,168.573,42.553,157.953
C00727=1032.294,39.392,407.716,168.571,42.554,157.953
C00728=1032.287,39.143,407.733,168.568,42.555,157.953
C00729=1032.281,38.893,407.749,168.566,42.556,157.953
C00730=1032.275,38.644,407.766,168.564,42.557,157.953
C00731=1032.269,38.394,407.782,168.561,42.558,157.953
C00732=1032.262,38.145,407.799,168.560,42.559,157.953
C00733=1032.256,37.896,407.815,168.557,42.560,157.953
C00734=1032.250,37.647,407.832,168.555,42.561,157.953
C00735=1032.244,37.396,407.848,168.552,42.562,157.953
C00736=1032.238,37.148,407.865,168.550,42.563,157.953
C00737=1032.231,36.899,407.881,168.547,42.564,157.953
C00738=1032.224,36.649,407.898,168.546,42.566,157.953
C00739=1032.218,36.399,407.914,168.543,42.567,157.953
C00740=1032.213,36.150,407.930,168.541,42.568,157.953
C00741=1032.206,35.901,407.946,168.538,42.569,157.953
C00742=1032.199,35.651,407.962,168.536,42.570,157.953
C00743=1032.193,35.402,407.979,168.534,42.571,157.953
C00744=1032.187,35.153,407.996,168.532,42.572,157.953
C00745=1032.180,34.904,408.011,168.529,42.574,157.953
C00746=1032.174,34.654,408.028,168.527,42.575,157.954
C00747=1032.168,34.404,408.044,168.524,42.576,157.954
C00748=1032.162,34.155,408.060,168.522,42.577,157.954
C00749=1032.155,33.906,408.076,168.521,42.578,157.954
C00750=1032.149,33.656,408.093,168.518,42.579,157.954
C00751=1032.143,33.407,408.109,168.516,42.580,157.954
C00752=1032.137,33.157,408.125,168.513,42.581,157.954
C00753=1032.130,32.908,408.141,168.511,42.582,157.954
C00754=1032.124,32.658,408.157,168.509,42.584,157.954
C00755=1032.118,32.409,408.174,168.507,42.585,157.954
C00756=1032.111,32.160,408.189,168.504,42.586,157.954
C00757=1032.105,31.910,408.206,168.502,42.587,157.954
C00758=1032.099,31.661,408.222,168.499,42.588,157.954
C00759=1032.092,31.411,408.238,168.497,42.589,157.954
C00760=1032.086,31.162,408.254,168.494,42.590,157.954
C00761=1032.080,30.913,408.270,168.493,42.591,157.954
C00762=1032.074,30.663,408.287,168.490,42.593,157.954
C00763=1032.068,30.414,408.303,168.488,42.594,157.954
C00764=1032.061,30.165,408.319,168.485,42.595,157.954
C00765=1032.055,29.915,408.335,168.483,42.596,157.954
C00766=1032.049,29.665,408.351,168.480,42.597,157.954
C00767=1032.042,29.416,408.367,168.479,42.598,157.954
C00768=1032.036,29.167,408.383,168.476,42.600,157.954
C00769=1032.030,28.918,408.400,168.474,42.601,157.955
C00770=1032.023,28.669,408.415,168.471,42.602,157.955
C00771=1032.017,28.382,408.435,168.468,42.603,157.955
C00772=1032.010,28.095,408.452,168.467,42.604,157.955
C00773=1032.002,27.809,408.471,168.464,42.605,157.955
C00774=1031.994,27.523,408.489,168.461,42.607,157.955
C00775=1031.988,27.274,408.505,168.458,42.608,157.955
C00776=1031.982,27.025,408.521,168.456,42.609,157.955
C00777=1031.976,26.775,408.537,168.453,42.610,157.955
C00778=1031.970,26.525,408.553,168.452,42.611,157.955
C00779=1031.963,26.276,408.569,168.449,42.612,157.955
C00780=1031.957,26.027,408.585,168.447,42.614,157.955
C00781=1031.951,25.778,408.600,168.444,42.615,157.955
C00782=1031.944,25.527,408.616,168.442,42.616,157.955
C00783=1031.938,25.278,408.632,168.440,42.617,157.955
C00784=1031.932,25.029,408.648,168.438,42.618,157.955
C00785=1031.925,24.780,408.664,168.435,42.619,157.955
C00786=1031.919,24.530,408.679,168.433,42.621,157.955
C00787=1031.913,24.281,408.695,168.430,42.622,157.955
C00788=1031.907,24.032,408.711,168.429,42.623,157.955
C00789=1031.900,23.783,408.727,168.426,42.624,157.955
C00790=1031.894,23.533,408.742,168.423,42.625,157.955
C00791=1031.888,23.284,408.758,168.421,42.626,157.955
C00792=1031.880,23.034,408.774,168.418,42.627,157.956
C00793=1031.875,22.784,408.790,168.416,42.629,157.956
C00794=1031.868,22.535,408.805,168.414,42.630,157.956
C00795=1031.862,22.285,408.822,168.412,42.631,157.956
C00796=1031.856,22.036,408.837,168.409,42.632,157.956
C00797=1031.850,21.786,408.853,168.407,42.633,157.956
C00798=1031.843,21.537,408.869,168.404,42.634,157.956
C00799=1031.837,21.287,408.884,168.402,42.635,157.956
C00800=1031.831,21.038,408.900,168.400,42.636,157.956
C00801=1031.825,20.789,408.916,168.398,42.637,157.956
C00802=1031.818,20.539,408.931,168.395,42.639,157.956
C00803=1031.812,20.290,408.947,168.393,42.640,157.956
C00804=1031.806,20.040,408.962,168.390,42.641,157.956
C00805=1031.799,19.791,408.978,168.388,42.642,157.956
C00806=1031.793,19.542,408.994,168.386,42.643,157.956
C00807=1031.787,19.292,409.009,168.383,42.644,157.956
C00808=1031.780,19.043,409.025,168.381,42.645,157.956
C00809=1031.775,18.793,409.040,168.378,42.647,157.956
C00810=1031.768,18.544,409.056,168.376,42.648,157.956
C00811=1031.762,18.295,409.071,168.374,42.649,157.956
C00812=1031.756,18.045,409.087,168.372,42.650,157.956
C00813=1031.749,17.796,409.102,168.369,42.651,157.956
C00814=1031.743,17.547,409.118,168.367,42.652,157.957
C00815=1031.737,17.297,409.133,168.364,42.654,157.957
C00816=1031.730,17.048,409.149,168.362,42.655,157.957
C00817=1031.724,16.798,409.164,168.360,42.656,157.957
C00818=1031.718,16.549,409.180,168.357,42.657,157.957
C00819=1031.712,16.299,409.195,168.355,42.658,157.957
C00820=1031.705,16.050,409.211,168.352,42.659,157.957
C00821=1031.699,15.800,409.226,168.350,42.661,157.957
C00822=1031.693,15.550,409.241,168.348,42.662,157.957
C00823=1031.686,15.301,409.257,168.346,42.663,157.957
C00824=1031.680,15.052,409.272,168.343,42.664,157.957
C00825=1031.674,14.802,409.288,168.340,42.666,157.957
C00826=1031.667,14.553,409.303,168.338,42.666,157.957
C00827=1031.661,14.303,409.319,168.335,42.668,157.957
C00828=1031.655,14.054,409.334,168.334,42.669,157.957
C00829=1031.649,13.804,409.349,168.331,42.670,157.957
C00830=1031.642,13.555,409.365,168.329,42.671,157.957
C00831=1031.636,13.305,409.380,168.326,42.673,157.957
C00832=1031.629,13.056,409.395,168.323,42.674,157.957
C00833=1031.623,12.806,409.410,168.322,42.675,157.958
C00834=1031.617,12.558,409.425,168.319,42.676,157.958
C00835=1031.609,12.272,409.443,168.316,42.678,157.958
C00836=1031.602,11.986,409.460,168.313,42.679,157.958
C00837=1031.595,11.702,409.477,168.310,42.681,157.958
C00838=1031.588,11.417,409.495,168.308,42.682,157.958
C00839=1031.581,11.167,409.510,168.306,42.683,157.958
C00840=1031.575,10.918,409.524,168.303,42.684,157.958
C00841=1031.569,10.669,409.540,168.300,42.686,157.958
C00842=1031.562,10.419,409.555,168.299,42.687,157.958
C00843=1031.556,10.170,409.570,168.296,42.688,157.958
C00844=1031.550,9.920,409.585,168.293,42.689,157.958
C00845=1031.543,9.670,409.600,168.291,42.691,157.958
C00846=1031.537,9.421,409.615,168.288,42.692,157.958
C00847=1031.530,9.172,409.630,168.287,42.693,157.958
C00848=1031.524,8.922,409.645,168.284,42.694,157.958
C00849=1031.518,8.673,409.660,168.281,42.696,157.958
C00850=1031.512,8.424,409.675,168.279,42.697,157.959
C00851=1031.505,8.174,409.690,168.276,42.698,157.959
C00852=1031.499,7.925,409.705,168.275,42.699,157.959
C00853=1031.492,7.675,409.720,168.272,42.701,157.959
C00854=1031.486,7.426,409.735,168.269,42.702,157.959
C00855=1031.479,7.176,409.750,168.267,42.703,157.959
C00856=1031.474,6.927,409.765,168.264,42.704,157.959
C00857=1031.467,6.677,409.780,168.262,42.706,157.959
C00858=1031.461,6.428,409.795,168.260,42.707,157.959
C00859=1031.454,6.178,409.810,168.257,42.708,157.959
C00860=1031.448,5.928,409.824,168.255,42.709,157.959
C00861=1031.441,5.679,409.840,168.252,42.710,157.959
C00862=1031.436,5.430,409.855,168.250,42.712,157.959
C00863=1031.429,5.181,409.870,168.248,42.713,157.959
C00864=1031.423,4.931,409.885,168.245,42.714,157.959
C00865=1031.416,4.681,409.900,168.243,42.715,157.959
C00866=1031.411,4.432,409.914,168.240,42.716,157.959
C00867=1031.404,4.183,409.929,168.238,42.718,157.959
C00868=1031.398,3.933,409.944,168.236,42.719,157.959
C00869=1031.391,3.683,409.959,168.233,42.720,157.959
C00870=1031.385,3.434,409.974,168.230,42.722,157.959
C00871=1031.379,3.185,409.989,168.228,42.723,157.960
C00872=1031.373,2.935,410.003,168.225,42.724,157.960
C00873=1031.367,2.685,410.018,168.224,42.725,157.960
C00874=1031.360,2.436,410.033,168.221,42.726,157.960
C00875=1031.354,2.187,410.048,168.218,42.728,157.960
C00876=1031.348,1.937,410.063,168.216,42.729,157.960
C00877=1031.342,1.688,410.078,168.213,42.730,157.960
C00878=1031.335,1.438,410.093,168.211,42.732,157.960
C00879=1031.329,1.189,410.107,168.209,42.733,157.960
C00880=1031.323,0.939,410.122,168.206,42.734,157.960
C00881=1031.317,0.690,410.137,168.204,42.735,157.960
C00882=1031.311,0.440,410.151,168.201,42.736,157.960
C00883=1031.305,0.190,410.166,168.198,42.737,157.960
C00884=1031.298,-0.059,410.181,168.197,42.739,157.960
C00885=1031.293,-0.308,410.196,168.194,42.740,157.960
C00886=1031.286,-0.558,410.211,168.191,42.741,157.960
C00887=1031.280,-0.808,410.225,168.189,42.742,157.960
C00888=1031.274,-1.057,410.240,168.186,42.743,157.960
C00889=1031.268,-1.306,410.255,168.184,42.744,157.960
C00890=1031.261,-1.556,410.270,168.182,42.745,157.960
C00891=1031.256,-1.805,410.284,168.179,42.747,157.960
C00892=1031.249,-2.055,410.298,168.177,42.748,157.960
C00893=1031.242,-2.304,410.313,168.174,42.749,157.960
C00894=1031.237,-2.553,410.328,168.171,42.750,157.960
C00895=1031.230,-2.803,410.343,168.170,42.751,157.961
C00896=1031.224,-3.053,410.358,168.167,42.752,157.961
C00897=1031.218,-3.302,410.371,168.165,42.753,157.961
C00898=1031.212,-3.552,410.386,168.162,42.755,157.961
C00899=1031.205,-3.835,410.403,168.159,42.756,157.961
C00900=1031.198,-4.118,410.419,168.156,42.757,157.961
C00901=1031.191,-4.401,410.436,168.154,42.759,157.961
C00902=1031.183,-4.684,410.452,168.151,42.760,157.961
C00903=1031.177,-4.934,410.466,168.148,42.762,157.961
C00904=1031.171,-5.183,410.481,168.145,42.763,157.961
C00905=1031.164,-5.433,410.495,168.144,42.764,157.961
C00906=1031.158,-5.682,410.510,168.141,42.766,157.961
C00907=1031.152,-5.931,410.524,168.138,42.767,157.961
C00908=1031.145,-6.181,410.538,168.136,42.768,157.961
C00909=1031.139,-6.430,410.552,168.134,42.770,157.961
C00910=1031.132,-6.680,410.567,168.131,42.771,157.961
C00911=1031.126,-6.930,410.581,168.128,42.772,157.961
C00912=1031.120,-7.179,410.596,168.126,42.774,157.962
C00913=1031.114,-7.429,410.609,168.123,42.775,157.962
C00914=1031.108,-7.678,410.624,168.120,42.776,157.962
C00915=1031.102,-7.928,410.638,168.119,42.778,157.962
C00916=1031.095,-8.177,410.652,168.116,42.779,157.962
C00917=1031.089,-8.426,410.667,168.113,42.780,157.962
C00918=1031.082,-8.676,410.681,168.110,42.781,157.962
C00919=1031.076,-8.925,410.695,168.109,42.783,157.962
C00920=1031.070,-9.176,410.709,168.106,42.784,157.962
C00921=1031.064,-9.424,410.723,168.103,42.785,157.962
C00922=1031.058,-9.674,410.738,168.101,42.787,157.962
C00923=1031.051,-9.924,410.752,168.098,42.788,157.962
C00924=1031.045,-10.173,410.766,168.096,42.789,157.962
C00925=1031.039,-10.423,410.781,168.093,42.790,157.962
C00926=1031.032,-10.672,410.794,168.091,42.792,157.962
C00927=1031.026,-10.922,410.809,168.088,42.793,157.962
C00928=1031.020,-11.171,410.822,168.085,42.794,157.962
C00929=1031.013,-11.421,410.837,168.084,42.796,157.962
C00930=1031.008,-11.670,410.851,168.081,42.797,157.962
C00931=1031.001,-11.920,410.865,168.078,42.798,157.962
C00932=1030.995,-12.169,410.879,168.075,42.799,157.962
C00933=1030.988,-12.419,410.894,168.074,42.801,157.963
C00934=1030.983,-12.668,410.908,168.071,42.802,157.963
C00935=1030.976,-12.918,410.921,168.068,42.803,157.963
C00936=1030.970,-13.167,410.936,168.066,42.804,157.963
C00937=1030.964,-13.417,410.950,168.063,42.806,157.963
C00938=1030.958,-13.666,410.964,168.060,42.807,157.963
C00939=1030.952,-13.916,410.978,168.058,42.808,157.963
C00940=1030.945,-14.166,410.991,168.056,42.809,157.963
C00941=1030.939,-14.415,411.006,168.053,42.811,157.963
C00942=1030.933,-14.665,411.020,168.050,42.812,157.963
C00943=1030.927,-14.915,411.034,168.048,42.813,157.963
C00944=1030.921,-15.164,411.048,168.046,42.815,157.963
C00945=1030.914,-15.414,411.062,168.043,42.816,157.963
C00946=1030.909,-15.663,411.076,168.040,42.818,157.963
C00947=1030.901,-15.913,411.090,168.038,42.819,157.963
C00948=1030.895,-16.162,411.104,168.036,42.820,157.963
C00949=1030.890,-16.412,411.117,168.033,42.822,157.963
C00950=1030.883,-16.662,411.131,168.030,42.823,157.964
C00951=1030.876,-16.910,411.145,168.027,42.824,157.964
C00952=1030.870,-17.160,411.159,168.025,42.825,157.964
C00953=1030.864,-17.410,411.173,168.023,42.827,157.964
C00954=1030.857,-17.660,411.186,168.020,42.828,157.964
C00955=1030.852,-17.909,411.200,168.017,42.830,157.964
C00956=1030.845,-18.159,411.214,168.015,42.831,157.964
C00957=1030.838,-18.408,411.228,168.012,42.832,157.964
C00958=1030.833,-18.657,411.242,168.010,42.834,157.964
C00959=1030.826,-18.907,411.255,168.007,42.835,157.964
C00960=1030.820,-19.157,411.268,168.004,42.837,157.964
C00961=1030.814,-19.407,411.283,168.002,42.838,157.964
C00962=1030.807,-19.656,411.297,168.000,42.839,157.964
C00963=1030.801,-19.937,411.312,167.997,42.841,157.964
C00964=1030.793,-20.218,411.327,167.994,42.842,157.964
C00965=1030.786,-20.501,411.342,167.990,42.844,157.964
C00966=1030.779,-20.782,411.358,167.987,42.845,157.964
C00967=1030.773,-21.031,411.371,167.985,42.847,157.965
C00968=1030.767,-21.281,411.386,167.983,42.848,157.965
C00969=1030.760,-21.530,411.399,167.980,42.849,157.965
C00970=1030.754,-21.780,411.412,167.977,42.851,157.965
C00971=1030.748,-22.030,411.426,167.975,42.852,157.965
C00972=1030.742,-22.279,411.440,167.973,42.853,157.965
C00973=1030.735,-22.528,411.454,167.970,42.855,157.965
C00974=1030.729,-22.778,411.467,167.967,42.856,157.965
C00975=1030.723,-23.027,411.481,167.964,42.857,157.965
C00976=1030.717,-23.277,411.494,167.962,42.859,157.965
C00977=1030.711,-23.526,411.508,167.960,42.860,157.965
C00978=1030.705,-23.776,411.522,167.957,42.861,157.965
C00979=1030.698,-24.026,411.535,167.954,42.863,157.965
C00980=1030.692,-24.275,411.548,167.952,42.864,157.965
C00981=1030.685,-24.525,411.562,167.949,42.866,157.965
C00982=1030.680,-24.774,411.576,167.947,42.867,157.965
C00983=1030.674,-25.024,411.589,167.944,42.868,157.965
C00984=1030.667,-25.274,411.603,167.941,42.870,157.965
C00985=1030.661,-25.523,411.617,167.939,42.871,157.965
C00986=1030.655,-25.772,411.630,167.936,42.873,157.965
C00987=1030.649,-26.022,411.642,167.934,42.874,157.966
C00988=1030.642,-26.272,411.656,167.931,42.875,157.966
C00989=1030.637,-26.522,411.670,167.928,42.876,157.966
C00990=1030.631,-26.771,411.683,167.926,42.878,157.966
C00991=1030.625,-27.020,411.696,167.923,42.879,157.966
C00992=1030.618,-27.270,411.710,167.921,42.880,157.966
C00993=1030.612,-27.520,411.723,167.918,42.882,157.966
C00994=1030.605,-27.769,411.737,167.916,42.883,157.966
C00995=1030.599,-28.019,411.749,167.913,42.885,157.966
C00996=1030.593,-28.269,411.763,167.910,42.886,157.966
C00997=1030.587,-28.518,411.777,167.907,42.888,157.966
C00998=1030.581,-28.768,411.790,167.906,42.889,157.966
C00999=1030.575,-29.017,411.803,167.903,42.890,157.966
C01000=1030.568,-29.267,411.816,167.900,42.892,157.966
C01001=1030.562,-29.517,411.829,167.897,42.893,157.966
C01002=1030.556,-29.766,411.843,167.895,42.895,157.967
C01003=1030.550,-30.015,411.856,167.892,42.896,157.967
C01004=1030.544,-30.265,411.869,167.889,42.898,157.967
C01005=1030.537,-30.515,411.882,167.886,42.899,157.967
C01006=1030.531,-30.764,411.895,167.885,42.901,157.967
C01007=1030.524,-31.014,411.909,167.882,42.902,157.967
C01008=1030.518,-31.263,411.921,167.879,42.904,157.967
C01009=1030.512,-31.513,411.935,167.876,42.905,157.967
C01010=1030.505,-31.763,411.948,167.873,42.906,157.967
C01011=1030.500,-32.013,411.961,167.871,42.908,157.967
C01012=1030.493,-32.262,411.974,167.868,42.909,157.967
C01013=1030.487,-32.511,411.987,167.866,42.911,157.967
C01014=1030.481,-32.761,412.000,167.863,42.912,157.967
C01015=1030.475,-33.010,412.013,167.861,42.914,157.967
C01016=1030.467,-33.260,412.026,167.858,42.915,157.967
C01017=1030.462,-33.510,412.039,167.855,42.917,157.968
C01018=1030.455,-33.759,412.052,167.852,42.918,157.967
C01019=1030.449,-34.009,412.064,167.849,42.919,157.967
C01020=1030.443,-34.258,412.078,167.847,42.921,157.968
C01021=1030.437,-34.507,412.091,167.845,42.922,157.968
C01022=1030.431,-34.757,412.104,167.842,42.924,157.968
C01023=1030.425,-35.007,412.117,167.839,42.925,157.968
C01024=1030.418,-35.257,412.130,167.837,42.927,157.968
C01025=1030.412,-35.506,412.143,167.834,42.928,157.968
C01026=1030.406,-35.756,412.156,167.831,42.929,157.968
C01027=1030.399,-36.036,412.170,167.828,42.931,157.968
C01028=1030.393,-36.317,412.186,167.826,42.933,157.968
C01029=1030.386,-36.598,412.200,167.823,42.934,157.968
C01030=1030.379,-36.879,412.214,167.819,42.936,157.968
C01031=1030.373,-37.128,412.228,167.816,42.937,157.968
C01032=1030.367,-37.378,412.240,167.815,42.939,157.968
C01033=1030.360,-37.627,412.253,167.812,42.940,157.968
C01034=1030.354,-37.877,412.266,167.809,42.941,157.968
C01035=1030.348,-38.126,412.279,167.806,42.943,157.969
C01036=1030.342,-38.376,412.292,167.803,42.944,157.969
C01037=1030.336,-38.626,412.305,167.801,42.946,157.969
C01038=1030.330,-38.876,412.318,167.798,42.947,157.969
C01039=1030.323,-39.124,412.330,167.795,42.949,157.969
C01040=1030.317,-39.374,412.343,167.792,42.950,157.969
C01041=1030.311,-39.624,412.356,167.791,42.952,157.969
C01042=1030.305,-39.873,412.368,167.788,42.953,157.969
C01043=1030.299,-40.123,412.381,167.785,42.955,157.969
C01044=1030.292,-40.372,412.394,167.782,42.956,157.969
C01045=1030.286,-40.622,412.406,167.780,42.958,157.969
C01046=1030.280,-40.872,412.418,167.777,42.960,157.969
C01047=1030.274,-41.121,412.432,167.774,42.961,157.969
C01048=1030.268,-41.371,412.444,167.772,42.963,157.969
C01049=1030.261,-41.620,412.456,167.769,42.964,157.969
C01050=1030.255,-41.870,412.469,167.766,42.966,157.970
C01051=1030.249,-42.120,412.482,167.763,42.967,157.970
C01052=1030.243,-42.370,412.494,167.760,42.969,157.970
C01053=1030.236,-42.619,412.506,167.758,42.970,157.970
C01054=1030.230,-42.868,412.520,167.755,42.972,157.970
C01055=1030.224,-43.118,412.532,167.752,42.973,157.970
C01056=1030.218,-43.368,412.544,167.749,42.975,157.970
C01057=1030.212,-43.618,412.557,167.747,42.976,157.970
C01058=1030.205,-43.867,412.570,167.744,42.978,157.970
C01059=1030.199,-44.117,412.582,167.742,42.979,157.970
C01060=1030.193,-44.366,412.595,167.739,42.980,157.970
C01061=1030.187,-44.616,412.607,167.737,42.982,157.970
C01062=1030.180,-44.866,412.619,167.734,42.983,157.970
C01063=1030.174,-45.115,412.632,167.731,42.985,157.970
C01064=1030.168,-45.365,412.645,167.728,42.986,157.970
C01065=1030.162,-45.615,412.657,167.726,42.988,157.971
C01066=1030.156,-45.864,412.669,167.723,42.989,157.971
C01067=1030.150,-46.114,412.682,167.720,42.991,157.971
C01068=1030.144,-46.363,412.694,167.717,42.992,157.971
C01069=1030.138,-46.612,412.707,167.715,42.994,157.971
C01070=1030.132,-46.862,412.719,167.712,42.996,157.971
C01071=1030.125,-47.112,412.731,167.709,42.997,157.971
C01072=1030.119,-47.362,412.744,167.707,42.999,157.971
C01073=1030.113,-47.612,412.756,167.704,43.000,157.971
C01074=1030.107,-47.861,412.768,167.701,43.002,157.971
C01075=1030.101,-48.110,412.781,167.698,43.003,157.971
C01076=1030.095,-48.360,412.793,167.696,43.005,157.971
C01077=1030.089,-48.610,412.805,167.693,43.006,157.971
C01078=1030.082,-48.859,412.818,167.690,43.008,157.971
C01079=1030.077,-49.109,412.831,167.688,43.009,157.971
C01080=1030.070,-49.359,412.843,167.686,43.011,157.972
C01081=1030.065,-49.608,412.855,167.683,43.012,157.972
C01082=1030.059,-49.858,412.868,167.680,43.014,157.972
C01083=1030.052,-50.107,412.880,167.677,43.015,157.972
C01084=1030.046,-50.357,412.892,167.674,43.017,157.972
C01085=1030.040,-50.607,412.905,167.672,43.018,157.972
C01086=1030.034,-50.857,412.917,167.669,43.020,157.972
C01087=1030.027,-51.107,412.928,167.666,43.022,157.972
C01088=1030.022,-51.356,412.940,167.663,43.023,157.972
C01089=1030.015,-51.606,412.952,167.661,43.025,157.972
C01090=1030.009,-51.855,412.964,167.658,43.027,157.972
C01091=1030.002,-52.136,412.978,167.654,43.029,157.972
C01092=1029.995,-52.417,412.991,167.652,43.031,157.973
C01093=1029.988,-52.699,413.005,167.648,43.033,157.973
C01094=1029.980,-52.979,413.018,167.645,43.034,157.973
C01095=1029.974,-53.229,413.031,167.643,43.036,157.973
C01096=1029.968,-53.479,413.043,167.640,43.037,157.973
C01097=1029.962,-53.728,413.053,167.637,43.039,157.973
C01098=1029.955,-53.978,413.065,167.635,43.041,157.973
C01099=1029.949,-54.228,413.078,167.632,43.043,157.973
C01100=1029.943,-54.477,413.090,167.628,43.044,157.973
C01101=1029.937,-54.727,413.101,167.625,43.046,157.973
C01102=1029.930,-54.976,413.113,167.623,43.048,157.973
C01103=1029.924,-55.226,413.125,167.620,43.050,157.974
C01104=1029.918,-55.476,413.137,167.617,43.051,157.974
C01105=1029.912,-55.725,413.148,167.615,43.053,157.974
C01106=1029.906,-55.975,413.161,167.612,43.055,157.974
C01107=1029.899,-56.225,413.173,167.609,43.056,157.974
C01108=1029.893,-56.474,413.185,167.606,43.058,157.974
C01109=1029.887,-56.724,413.195,167.604,43.059,157.974
C01110=1029.881,-56.974,413.208,167.601,43.061,157.974
C01111=1029.874,-57.223,413.220,167.598,43.063,157.974
C01112=1029.868,-57.473,413.231,167.596,43.064,157.974
C01113=1029.862,-57.722,413.243,167.593,43.066,157.974
C01114=1029.856,-57.972,413.255,167.590,43.068,157.974
C01115=1029.850,-58.222,413.267,167.587,43.069,157.974
C01116=1029.844,-58.471,413.278,167.585,43.071,157.975
C01117=1029.837,-58.721,413.290,167.581,43.073,157.975
C01118=1029.832,-58.971,413.302,167.578,43.075,157.975
C01119=1029.825,-59.220,413.314,167.576,43.076,157.975
C01120=1029.819,-59.470,413.326,167.573,43.078,157.975
C01121=1029.812,-59.720,413.337,167.570,43.080,157.975
C01122=1029.806,-59.969,413.348,167.567,43.081,157.975
C01123=1029.801,-60.219,413.360,167.565,43.083,157.975
C01124=1029.794,-60.469,413.372,167.562,43.085,157.975
C01125=1029.788,-60.718,413.384,167.559,43.087,157.975
C01126=1029.782,-60.968,413.395,167.557,43.088,157.975
C01127=1029.776,-61.218,413.408,167.554,43.090,157.976
C01128=1029.770,-61.467,413.418,167.551,43.091,157.976
C01129=1029.764,-61.717,413.430,167.548,43.093,157.976
C01130=1029.758,-61.966,413.441,167.546,43.094,157.976
C01131=1029.752,-62.216,413.454,167.543,43.096,157.976
C01132=1029.746,-62.467,413.465,167.540,43.098,157.976
C01133=1029.739,-62.715,413.477,167.537,43.099,157.976
C01134=1029.733,-62.966,413.488,167.534,43.101,157.976
C01135=1029.727,-63.214,413.499,167.531,43.103,157.976
C01136=1029.721,-63.465,413.511,167.528,43.104,157.976
C01137=1029.715,-63.714,413.523,167.526,43.106,157.976
C01138=1029.709,-63.964,413.534,167.523,43.108,157.976
C01139=1029.702,-64.214,413.546,167.520,43.110,157.977
C01140=1029.697,-64.463,413.557,167.518,43.111,157.977
C01141=1029.691,-64.713,413.570,167.515,43.113,157.977
C01142=1029.685,-64.962,413.580,167.512,43.115,157.977
C01143=1029.678,-65.212,413.592,167.509,43.116,157.977
C01144=1029.673,-65.461,413.603,167.507,43.118,157.977
C01145=1029.666,-65.712,413.615,167.504,43.120,157.977
C01146=1029.661,-65.961,413.627,167.501,43.121,157.977
C01147=1029.655,-66.211,413.638,167.498,43.123,157.977
C01148=1029.649,-66.460,413.650,167.495,43.125,157.977
C01149=1029.642,-66.710,413.661,167.492,43.127,157.977
C01150=1029.637,-66.960,413.672,167.489,43.128,157.977
C01151=1029.631,-67.209,413.684,167.487,43.130,157.977
C01152=1029.625,-67.459,413.695,167.484,43.131,157.978
C01153=1029.619,-67.709,413.706,167.481,43.133,157.977
C01154=1029.613,-67.958,413.718,167.479,43.134,157.978
C01155=1029.606,-68.241,413.731,167.475,43.136,157.978
C01156=1029.600,-68.523,413.744,167.472,43.138,157.978
C01157=1029.592,-68.805,413.756,167.469,43.140,157.978
C01158=1029.585,-69.088,413.769,167.466,43.142,157.978
C01159=1029.579,-69.337,413.781,167.463,43.143,157.978
C01160=1029.574,-69.587,413.792,167.460,43.145,157.978
C01161=1029.568,-69.837,413.803,167.458,43.147,157.978
C01162=1029.562,-70.087,413.815,167.455,43.148,157.978
C01163=1029.556,-70.336,413.826,167.452,43.150,157.978
C01164=1029.550,-70.585,413.837,167.450,43.152,157.978
C01165=1029.544,-70.835,413.848,167.446,43.153,157.978
C01166=1029.539,-71.085,413.860,167.443,43.155,157.979
C01167=1029.532,-71.335,413.872,167.440,43.157,157.979
C01168=1029.526,-71.584,413.883,167.437,43.158,157.979
C01169=1029.520,-71.834,413.893,167.435,43.160,157.979
C01170=1029.514,-72.084,413.905,167.432,43.162,157.979
C01171=1029.508,-72.333,413.916,167.429,43.163,157.979
C01172=1029.502,-72.582,413.927,167.427,43.165,157.979
C01173=1029.497,-72.833,413.939,167.424,43.167,157.979
C01174=1029.491,-73.082,413.950,167.421,43.168,157.979
C01175=1029.485,-73.332,413.961,167.418,43.170,157.979
C01176=1029.479,-73.582,413.972,167.416,43.172,157.979
C01177=1029.473,-73.831,413.983,167.412,43.173,157.979
C01178=1029.467,-74.081,413.994,167.409,43.175,157.979
C01179=1029.461,-74.330,414.006,167.407,43.177,157.979
C01180=1029.455,-74.580,414.017,167.404,43.179,157.980
C01181=1029.449,-74.829,414.027,167.401,43.180,157.980
C01182=1029.443,-75.080,414.039,167.398,43.182,157.980
C01183=1029.437,-75.329,414.050,167.396,43.183,157.980
C01184=1029.431,-75.579,414.060,167.393,43.185,157.980
C01185=1029.425,-75.829,414.072,167.389,43.187,157.980
C01186=1029.419,-76.078,414.082,167.387,43.189,157.980
C01187=1029.413,-76.327,414.093,167.384,43.191,157.980
C01188=1029.407,-76.578,414.104,167.381,43.193,157.980
C01189=1029.401,-76.828,414.114,167.379,43.194,157.980
C01190=1029.395,-77.077,414.125,167.376,43.196,157.980
C01191=1029.389,-77.327,414.136,167.372,43.198,157.981
C01192=1029.383,-77.577,414.147,167.370,43.200,157.981
C01193=1029.377,-77.826,414.158,167.367,43.202,157.981
C01194=1029.371,-78.076,414.168,167.364,43.204,157.981
C01195=1029.365,-78.326,414.180,167.362,43.205,157.981
C01196=1029.359,-78.575,414.191,167.359,43.207,157.981
C01197=1029.353,-78.825,414.201,167.356,43.208,157.981
C01198=1029.347,-79.075,414.213,167.352,43.211,157.981
C01199=1029.340,-79.324,414.223,167.350,43.212,157.981
C01200=1029.335,-79.574,414.233,167.347,43.214,157.981
C01201=1029.329,-79.824,414.244,167.345,43.216,157.982
C01202=1029.323,-80.074,414.255,167.342,43.218,157.982
C01203=1029.317,-80.323,414.266,167.338,43.220,157.982
C01204=1029.311,-80.573,414.276,167.336,43.222,157.982
C01205=1029.305,-80.823,414.287,167.333,43.224,157.982
C01206=1029.298,-81.073,414.297,167.330,43.226,157.982
C01207=1029.292,-81.322,414.308,167.328,43.227,157.982
C01208=1029.287,-81.572,414.319,167.324,43.229,157.982
C01209=1029.281,-81.821,414.328,167.321,43.231,157.982
C01210=1029.274,-82.072,414.340,167.319,43.233,157.982
C01211=1029.268,-82.321,414.350,167.316,43.235,157.983
C01212=1029.262,-82.571,414.360,167.312,43.237,157.983
C01213=1029.257,-82.820,414.371,167.310,43.239,157.983
C01214=1029.250,-83.069,414.381,167.307,43.241,157.983
C01215=1029.244,-83.320,414.392,167.304,43.243,157.983
C01216=1029.238,-83.569,414.402,167.302,43.245,157.983
C01217=1029.232,-83.819,414.413,167.298,43.247,157.983
C01218=1029.226,-84.069,414.423,167.295,43.248,157.983
C01219=1029.219,-84.353,414.435,167.292,43.250,157.983
C01220=1029.212,-84.637,414.447,167.289,43.253,157.984
C01221=1029.205,-84.922,414.459,167.285,43.255,157.984
C01222=1029.198,-85.207,414.471,167.282,43.257,157.984
C01223=1029.192,-85.457,414.481,167.279,43.259,157.984
C01224=1029.187,-85.706,414.491,167.276,43.261,157.984
C01225=1029.180,-85.955,414.502,167.274,43.263,157.984
C01226=1029.175,-86.205,414.512,167.271,43.265,157.984
C01227=1029.168,-86.454,414.522,167.268,43.267,157.984
C01228=1029.162,-86.705,414.533,167.265,43.268,157.984
C01229=1029.156,-86.954,414.543,167.262,43.270,157.984
C01230=1029.150,-87.205,414.553,167.260,43.272,157.985
C01231=1029.144,-87.454,414.564,167.256,43.274,157.985
C01232=1029.138,-87.704,414.574,167.253,43.276,157.985
C01233=1029.133,-87.953,414.585,167.251,43.278,157.985
C01234=1029.126,-88.203,414.594,167.248,43.280,157.985
C01235=1029.121,-88.453,414.605,167.245,43.282,157.985
C01236=1029.115,-88.702,414.615,167.242,43.284,157.985
C01237=1029.109,-88.952,414.625,167.239,43.286,157.985
C01238=1029.103,-89.202,414.635,167.236,43.288,157.985
C01239=1029.097,-89.451,414.646,167.234,43.289,157.986
C01240=1029.091,-89.701,414.655,167.230,43.291,157.986
C01241=1029.085,-89.950,414.666,167.227,43.293,157.986
C01242=1029.080,-90.201,414.676,167.225,43.295,157.986
C01243=1029.072,-90.450,414.687,167.222,43.297,157.986
C01244=1029.067,-90.701,414.697,167.219,43.299,157.986
C01245=1029.061,-90.950,414.707,167.216,43.301,157.986
C01246=1029.055,-91.200,414.718,167.213,43.303,157.986
C01247=1029.049,-91.450,414.727,167.210,43.305,157.986
C01248=1029.043,-91.699,414.738,167.208,43.307,157.986
C01249=1029.037,-91.949,414.748,167.204,43.309,157.987
C01250=1029.032,-92.199,414.758,167.201,43.310,157.987
C01251=1029.026,-92.448,414.768,167.199,43.312,157.987
C01252=1029.020,-92.698,414.778,167.196,43.314,157.987
C01253=1029.014,-92.947,414.788,167.192,43.316,157.987
C01254=1029.008,-93.197,414.798,167.190,43.318,157.987
C01255=1029.002,-93.447,414.808,167.187,43.320,157.987
C01256=1028.997,-93.697,414.818,167.184,43.322,157.987
C01257=1028.990,-93.946,414.828,167.182,43.324,157.987
C01258=1028.985,-94.196,414.839,167.178,43.326,157.987
C01259=1028.979,-94.446,414.848,167.175,43.328,157.988
C01260=1028.973,-94.695,414.859,167.173,43.330,157.988
C01261=1028.967,-94.945,414.869,167.170,43.331,157.988
C01262=1028.961,-95.195,414.879,167.166,43.333,157.988
C01263=1028.955,-95.445,414.888,167.164,43.335,157.988
C01264=1028.949,-95.695,414.899,167.161,43.337,157.988
C01265=1028.943,-95.944,414.909,167.158,43.339,157.988
C01266=1028.938,-96.194,414.919,167.156,43.341,157.988
C01267=1028.932,-96.444,414.928,167.152,43.343,157.988
C01268=1028.927,-96.694,414.938,167.149,43.345,157.988
C01269=1028.920,-96.943,414.949,167.147,43.347,157.989
C01270=1028.915,-97.193,414.959,167.144,43.349,157.989
C01271=1028.909,-97.443,414.968,167.140,43.351,157.989
C01272=1028.903,-97.693,414.978,167.138,43.353,157.989
C01273=1028.897,-97.943,414.988,167.135,43.355,157.989
C01274=1028.892,-98.192,414.997,167.133,43.357,157.989
C01275=1028.885,-98.442,415.007,167.129,43.359,157.989
C01276=1028.880,-98.692,415.017,167.126,43.361,157.989
C01277=1028.873,-98.941,415.027,167.124,43.363,157.989
C01278=1028.867,-99.191,415.037,167.120,43.366,157.990
C01279=1028.861,-99.441,415.046,167.118,43.367,157.990
C01280=1028.856,-99.691,415.057,167.115,43.369,157.990
C01281=1028.850,-99.940,415.066,167.112,43.371,157.990
C01282=1028.844,-100.190,415.075,167.109,43.373,157.990
C01283=1028.837,-100.476,415.086,167.105,43.376,157.990
C01284=1028.830,-100.763,415.097,167.103,43.378,157.990
C01285=1028.823,-101.050,415.108,167.099,43.381,157.991
C01286=1028.816,-101.337,415.119,167.095,43.383,157.991
C01287=1028.811,-101.587,415.129,167.093,43.385,157.991
C01288=1028.805,-101.836,415.139,167.090,43.387,157.991
C01289=1028.799,-102.086,415.148,167.087,43.389,157.991
C01290=1028.793,-102.335,415.158,167.084,43.391,157.991
C01291=1028.787,-102.585,415.167,167.081,43.393,157.991
C01292=1028.782,-102.835,415.177,167.078,43.395,157.991
C01293=1028.776,-103.084,415.187,167.075,43.398,157.992
C01294=1028.770,-103.334,415.196,167.073,43.399,157.992
C01295=1028.764,-103.584,415.206,167.069,43.401,157.992
C01296=1028.758,-103.833,415.215,167.066,43.403,157.992
C01297=1028.753,-104.083,415.225,167.064,43.405,157.992
C01298=1028.747,-104.334,415.234,167.061,43.407,157.992
C01299=1028.741,-104.583,415.243,167.057,43.410,157.992
C01300=1028.735,-104.833,415.253,167.055,43.412,157.992
C01301=1028.729,-105.082,415.262,167.052,43.414,157.992
C01302=1028.723,-105.332,415.272,167.048,43.416,157.993
C01303=1028.717,-105.582,415.282,167.046,43.418,157.993
C01304=1028.712,-105.832,415.290,167.043,43.420,157.993
C01305=1028.706,-106.082,415.300,167.041,43.422,157.993
C01306=1028.700,-106.332,415.310,167.037,43.424,157.993
C01307=1028.694,-106.581,415.319,167.034,43.426,157.993
C01308=1028.688,-106.830,415.328,167.032,43.428,157.993
C01309=1028.682,-107.081,415.337,167.028,43.431,157.993
C01310=1028.676,-107.330,415.346,167.026,43.432,157.994
C01311=1028.671,-107.580,415.357,167.023,43.434,157.994
C01312=1028.665,-107.830,415.366,167.019,43.436,157.994
C01313=1028.660,-108.080,415.375,167.017,43.439,157.994
C01314=1028.653,-108.329,415.384,167.014,43.441,157.994
C01315=1028.647,-108.579,415.394,167.010,43.443,157.994
C01316=1028.642,-108.829,415.402,167.008,43.445,157.994
C01317=1028.636,-109.079,415.412,167.005,43.447,157.994
C01318=1028.630,-109.329,415.421,167.002,43.449,157.995
C01319=1028.624,-109.578,415.430,166.999,43.452,157.995
C01320=1028.618,-109.828,415.439,166.997,43.454,157.995
C01321=1028.612,-110.078,415.449,166.993,43.456,157.995
C01322=1028.607,-110.328,415.457,166.990,43.458,157.995
C01323=1028.601,-110.577,415.467,166.988,43.460,157.995
C01324=1028.595,-110.827,415.475,166.984,43.462,157.995
C01325=1028.588,-111.077,415.485,166.982,43.464,157.995
C01326=1028.582,-111.326,415.494,166.979,43.467,157.996
C01327=1028.577,-111.576,415.503,166.975,43.469,157.996
C01328=1028.571,-111.826,415.512,166.973,43.471,157.996
C01329=1028.566,-112.076,415.521,166.970,43.473,157.996
C01330=1028.559,-112.325,415.530,166.967,43.476,157.996
C01331=1028.554,-112.576,415.539,166.964,43.477,157.996
C01332=1028.548,-112.825,415.548,166.961,43.479,157.996
C01333=1028.542,-113.075,415.558,166.958,43.482,157.997
C01334=1028.537,-113.324,415.566,166.955,43.484,157.997
C01335=1028.530,-113.574,415.576,166.953,43.486,157.997
C01336=1028.525,-113.824,415.584,166.949,43.489,157.997
C01337=1028.519,-114.074,415.594,166.946,43.490,157.997
C01338=1028.514,-114.323,415.602,166.944,43.492,157.997
C01339=1028.507,-114.573,415.612,166.940,43.495,157.997
C01340=1028.502,-114.823,415.620,166.938,43.497,157.997
C01341=1028.496,-115.073,415.629,166.935,43.499,157.998
C01342=1028.490,-115.322,415.638,166.932,43.502,157.998
C01343=1028.484,-115.573,415.647,166.929,43.504,157.998
C01344=1028.479,-115.822,415.656,166.926,43.506,157.998
C01345=1028.473,-116.072,415.665,166.923,43.508,157.998
C01346=1028.467,-116.322,415.673,166.920,43.510,157.998
C01347=1028.458,-116.717,415.687,166.916,43.514,157.998
C01348=1028.448,-117.112,415.701,166.911,43.517,157.999
C01349=1028.440,-117.507,415.716,166.906,43.521,157.999
C01350=1028.430,-117.902,415.730,166.902,43.524,157.999
C01351=1028.425,-118.152,415.738,166.898,43.527,157.999
C01352=1028.419,-118.402,415.748,166.896,43.529,157.999
C01353=1028.413,-118.651,415.756,166.893,43.531,158.000
C01354=1028.407,-118.901,415.764,166.890,43.533,158.000
C01355=1028.402,-119.151,415.773,166.887,43.535,158.000
C01356=1028.396,-119.401,415.782,166.884,43.538,158.000
C01357=1028.389,-119.651,415.790,166.881,43.540,158.000
C01358=1028.384,-119.900,415.799,166.878,43.542,158.000
C01359=1028.378,-120.151,415.808,166.876,43.544,158.000
C01360=1028.373,-120.400,415.817,166.872,43.546,158.000
C01361=1028.367,-120.649,415.825,166.870,43.549,158.001
C01362=1028.361,-120.900,415.834,166.867,43.551,158.001
C01363=1028.356,-121.149,415.842,166.863,43.554,158.001
C01364=1028.350,-121.398,415.851,166.861,43.556,158.001
C01365=1028.343,-121.649,415.860,166.857,43.558,158.001
C01366=1028.338,-121.898,415.868,166.855,43.560,158.001
C01367=1028.332,-122.149,415.877,166.852,43.562,158.001
C01368=1028.327,-122.398,415.885,166.849,43.565,158.002
C01369=1028.321,-122.648,415.893,166.846,43.567,158.002
C01370=1028.315,-122.898,415.903,166.843,43.569,158.002
C01371=1028.310,-123.147,415.911,166.840,43.571,158.002
C01372=1028.304,-123.397,415.920,166.837,43.574,158.002
C01373=1028.298,-123.647,415.928,166.835,43.576,158.002
C01374=1028.292,-123.897,415.937,166.831,43.579,158.003
C01375=1028.287,-124.147,415.945,166.829,43.581,158.003
C01376=1028.281,-124.397,415.953,166.825,43.583,158.003
C01377=1028.275,-124.646,415.962,166.822,43.585,158.003
C01378=1028.270,-124.896,415.970,166.820,43.587,158.003
C01379=1028.263,-125.146,415.979,166.816,43.590,158.003
C01380=1028.258,-125.396,415.987,166.814,43.593,158.003
C01381=1028.252,-125.645,415.995,166.810,43.595,158.004
C01382=1028.246,-125.896,416.004,166.808,43.597,158.004
C01383=1028.241,-126.146,416.012,166.805,43.599,158.004
C01384=1028.235,-126.395,416.020,166.802,43.602,158.004
C01385=1028.230,-126.645,416.029,166.799,43.604,158.004
C01386=1028.223,-126.895,416.037,166.797,43.606,158.004
C01387=1028.218,-127.144,416.045,166.793,43.608,158.004
C01388=1028.212,-127.394,416.053,166.790,43.611,158.005
C01389=1028.207,-127.644,416.062,166.787,43.613,158.005
C01390=1028.201,-127.894,416.071,166.784,43.616,158.005
C01391=1028.196,-128.142,416.079,166.782,43.618,158.005
C01392=1028.191,-128.392,416.089,166.779,43.619,158.005
C01393=1028.186,-128.642,416.098,166.776,43.620,158.005
C01394=1028.183,-128.892,416.109,166.773,43.621,158.005
C01395=1028.180,-129.153,416.121,166.771,43.621,158.005
C01396=1028.178,-129.415,416.132,166.768,43.620,158.004
C01397=1028.176,-129.677,416.145,166.766,43.619,158.004
C01398=1028.175,-129.939,416.159,166.763,43.618,158.004
C01399=1028.175,-130.189,416.172,166.762,43.616,158.003
C01400=1028.175,-130.439,416.186,166.759,43.613,158.002
C01401=1028.175,-130.688,416.201,166.757,43.611,158.002
C01402=1028.177,-130.937,416.216,166.756,43.607,158.001
C01403=1028.180,-131.317,416.241,166.753,43.601,158.000
C01404=1028.184,-131.697,416.266,166.751,43.594,157.999
C01405=1028.191,-132.075,416.293,166.749,43.587,157.997
C01406=1028.199,-132.453,416.321,166.746,43.578,157.995
C01407=1027.885,-132.479,416.008,166.698,43.829,158.033
C01408=1027.881,-132.229,415.989,166.699,43.834,158.034
C01409=1027.877,-131.979,415.971,166.701,43.840,158.035
C01410=1027.873,-131.729,415.953,166.702,43.846,158.037
C01411=1027.869,-131.479,415.936,166.704,43.850,158.037
C01412=1027.867,-131.230,415.920,166.705,43.855,158.038
C01413=1027.865,-130.979,415.904,166.708,43.859,158.039
C01414=1027.864,-130.729,415.888,166.708,43.861,158.040
C01415=1027.862,-130.480,415.874,166.710,43.865,158.040
C01416=1027.863,-130.230,415.859,166.713,43.867,158.041
C01417=1027.863,-129.980,415.846,166.715,43.869,158.042
C01418=1027.863,-129.730,415.833,166.718,43.870,158.042
C01419=1027.865,-129.480,415.820,166.720,43.871,158.042
C01420=1027.867,-129.230,415.809,166.722,43.871,158.043
C01421=1027.870,-128.981,415.797,166.725,43.872,158.043
C01422=1027.874,-128.732,415.787,166.727,43.871,158.043
C01423=1027.878,-128.481,415.777,166.729,43.870,158.043
C01424=1027.882,-128.232,415.767,166.732,43.869,158.043
C01425=1027.887,-127.982,415.758,166.735,43.867,158.043
C01426=1027.892,-127.733,415.750,166.739,43.865,158.043
C01427=1027.898,-127.483,415.742,166.741,43.862,158.043
C01428=1027.904,-127.233,415.733,166.744,43.860,158.043
C01429=1027.910,-126.984,415.726,166.747,43.858,158.042
C01430=1027.915,-126.734,415.717,166.750,43.855,158.042
C01431=1027.921,-126.485,415.709,166.753,43.853,158.042
C01432=1027.927,-126.234,415.700,166.756,43.850,158.042
C01433=1027.932,-125.984,415.692,166.759,43.848,158.042
C01434=1027.938,-125.735,415.684,166.762,43.846,158.042
C01435=1027.944,-125.485,415.675,166.764,43.844,158.041
C01436=1027.950,-125.235,415.667,166.768,43.841,158.041
C01437=1027.955,-124.985,415.659,166.770,43.838,158.041
C01438=1027.961,-124.736,415.651,166.774,43.836,158.041
C01439=1027.967,-124.486,415.642,166.776,43.834,158.041
C01440=1027.972,-124.236,415.633,166.779,43.832,158.041
C01441=1027.978,-123.987,415.626,166.782,43.829,158.041
C01442=1027.984,-123.736,415.617,166.785,43.827,158.040
C01443=1027.989,-123.486,415.608,166.789,43.824,158.040
C01444=1027.995,-123.237,415.600,166.791,43.822,158.040
C01445=1028.001,-122.987,415.591,166.794,43.820,158.040
C01446=1028.007,-122.737,415.582,166.797,43.817,158.040
C01447=1028.012,-122.488,415.574,166.800,43.816,158.040
C01448=1028.019,-122.238,415.566,166.803,43.813,158.040
C01449=1028.024,-121.988,415.557,166.806,43.811,158.039
C01450=1028.029,-121.738,415.549,166.808,43.808,158.039
C01451=1028.035,-121.488,415.540,166.812,43.806,158.039
C01452=1028.041,-121.239,415.531,166.815,43.804,158.039
C01453=1028.047,-120.989,415.522,166.817,43.802,158.039
C01454=1028.052,-120.739,415.514,166.821,43.799,158.039
C01455=1028.058,-120.489,415.505,166.823,43.797,158.039
C01456=1028.064,-120.239,415.497,166.827,43.794,158.038
C01457=1028.070,-119.990,415.488,166.829,43.792,158.038
C01458=1028.076,-119.740,415.479,166.832,43.790,158.038
C01459=1028.081,-119.490,415.471,166.835,43.788,158.038
C01460=1028.087,-119.240,415.463,166.838,43.785,158.038
C01461=1028.093,-118.991,415.453,166.842,43.783,158.038
C01462=1028.098,-118.741,415.445,166.844,43.781,158.038
C01463=1028.104,-118.490,415.436,166.847,43.778,158.037
C01464=1028.110,-118.241,415.427,166.850,43.776,158.037
C01465=1028.116,-117.992,415.419,166.853,43.774,158.037
C01466=1028.122,-117.742,415.410,166.855,43.772,158.037
C01467=1028.127,-117.492,415.401,166.859,43.769,158.037
C01468=1028.134,-117.206,415.391,166.862,43.767,158.037
C01469=1028.141,-116.920,415.381,166.866,43.764,158.037
C01470=1028.147,-116.633,415.371,166.868,43.761,158.036
C01471=1028.154,-116.347,415.360,166.872,43.759,158.036
C01472=1028.159,-116.098,415.351,166.875,43.757,158.036
C01473=1028.166,-115.848,415.343,166.878,43.754,158.036
C01474=1028.171,-115.598,415.335,166.881,43.752,158.036
C01475=1028.177,-115.348,415.325,166.884,43.750,158.036
C01476=1028.183,-115.098,415.316,166.887,43.747,158.036
C01477=1028.189,-114.849,415.307,166.890,43.745,158.036
C01478=1028.194,-114.599,415.298,166.893,43.743,158.035
C01479=1028.200,-114.348,415.290,166.895,43.741,158.035
C01480=1028.209,-113.990,415.277,166.900,43.738,158.035
C01481=1028.217,-113.632,415.264,166.904,43.734,158.035
C01482=1028.225,-113.272,415.251,166.909,43.731,158.035
C01483=1028.233,-112.914,415.238,166.913,43.728,158.034
C01484=1028.239,-112.665,415.229,166.915,43.726,158.034
C01485=1028.245,-112.414,415.220,166.918,43.724,158.034
C01486=1028.250,-112.165,415.211,166.922,43.721,158.034
C01487=1028.256,-111.915,415.202,166.924,43.719,158.034
C01488=1028.262,-111.665,415.192,166.927,43.717,158.034
C01489=1028.268,-111.415,415.184,166.930,43.714,158.034
C01490=1028.274,-111.166,415.174,166.933,43.713,158.034
C01491=1028.279,-110.916,415.165,166.936,43.711,158.033
C01492=1028.285,-110.666,415.156,166.939,43.708,158.033
C01493=1028.291,-110.416,415.147,166.942,43.706,158.033
C01494=1028.297,-110.166,415.138,166.945,43.704,158.033
C01495=1028.303,-109.917,415.129,166.948,43.701,158.033
C01496=1028.308,-109.668,415.119,166.950,43.699,158.033
C01497=1028.314,-109.417,415.111,166.954,43.697,158.033
C01498=1028.321,-109.167,415.101,166.957,43.695,158.032
C01499=1028.326,-108.918,415.092,166.959,43.693,158.032
C01500=1028.332,-108.668,415.083,166.963,43.691,158.032
C01501=1028.338,-108.418,415.073,166.965,43.688,158.032
C01502=1028.343,-108.168,415.065,166.968,43.686,158.032
C01503=1028.350,-107.919,415.055,166.972,43.684,158.032
C01504=1028.355,-107.669,415.046,166.974,43.681,158.032
C01505=1028.361,-107.419,415.037,166.977,43.680,158.032
C01506=1028.367,-107.169,415.028,166.980,43.678,158.032
C01507=1028.373,-106.919,415.018,166.983,43.675,158.031
C01508=1028.379,-106.670,415.009,166.985,43.673,158.031
C01509=1028.385,-106.420,415.000,166.989,43.671,158.031
C01510=1028.391,-106.170,414.990,166.992,43.669,158.031
C01511=1028.397,-105.921,414.981,166.994,43.666,158.031
C01512=1028.402,-105.671,414.971,166.998,43.664,158.031
C01513=1028.408,-105.421,414.962,167.000,43.662,158.031
C01514=1028.413,-105.171,414.953,167.003,43.661,158.031
C01515=1028.420,-104.922,414.943,167.007,43.658,158.030
C01516=1028.426,-104.672,414.934,167.009,43.656,158.030
C01517=1028.431,-104.423,414.925,167.012,43.654,158.030
C01518=1028.437,-104.173,414.915,167.016,43.652,158.030
C01519=1028.443,-103.923,414.905,167.018,43.649,158.030
C01520=1028.449,-103.673,414.895,167.021,43.647,158.030
C01521=1028.454,-103.423,414.887,167.024,43.645,158.030
C01522=1028.461,-103.174,414.877,167.027,43.643,158.030
C01523=1028.467,-102.924,414.868,167.030,43.642,158.029
C01524=1028.472,-102.674,414.858,167.033,43.639,158.029
C01525=1028.478,-102.425,414.848,167.036,43.637,158.029
C01526=1028.484,-102.175,414.839,167.038,43.635,158.029
C01527=1028.490,-101.925,414.829,167.041,43.633,158.029
C01528=1028.495,-101.711,414.821,167.044,43.631,158.029
C01529=1028.500,-101.498,414.812,167.046,43.629,158.029
C01530=1028.505,-101.284,414.805,167.049,43.627,158.029
C01531=1028.509,-101.070,414.797,167.052,43.625,158.029
C01532=1028.515,-100.857,414.788,167.054,43.624,158.028
C01533=1028.520,-100.643,414.780,167.057,43.622,158.028
C01534=1028.525,-100.429,414.772,167.058,43.620,158.028
C01535=1028.530,-100.216,414.763,167.061,43.618,158.028
C01536=1028.536,-99.965,414.753,167.065,43.616,158.028
C01537=1028.541,-99.716,414.744,167.067,43.614,158.028
C01538=1028.548,-99.467,414.735,167.070,43.612,158.028
C01539=1028.554,-99.217,414.725,167.073,43.610,158.028
C01540=1028.560,-98.967,414.715,167.076,43.608,158.028
C01541=1028.565,-98.717,414.705,167.079,43.606,158.027
C01542=1028.572,-98.467,414.696,167.081,43.604,158.027
C01543=1028.577,-98.218,414.686,167.085,43.602,158.027
C01544=1028.583,-97.968,414.677,167.088,43.599,158.027
C01545=1028.589,-97.718,414.667,167.090,43.597,158.027
C01546=1028.595,-97.468,414.657,167.094,43.595,158.027
C01547=1028.600,-97.218,414.647,167.097,43.593,158.027
C01548=1028.607,-96.969,414.637,167.099,43.591,158.027
C01549=1028.612,-96.719,414.627,167.102,43.589,158.027
C01550=1028.618,-96.469,414.617,167.105,43.587,158.026
C01551=1028.624,-96.220,414.608,167.108,43.585,158.026
C01552=1028.629,-95.970,414.598,167.111,43.584,158.026
C01553=1028.636,-95.721,414.587,167.113,43.582,158.026
C01554=1028.641,-95.471,414.577,167.117,43.580,158.026
C01555=1028.648,-95.221,414.568,167.120,43.578,158.026
C01556=1028.653,-94.971,414.557,167.122,43.576,158.026
C01557=1028.659,-94.722,414.547,167.125,43.574,158.026
C01558=1028.665,-94.471,414.537,167.129,43.572,158.026
C01559=1028.671,-94.222,414.527,167.131,43.569,158.025
C01560=1028.676,-93.972,414.518,167.134,43.567,158.025
C01561=1028.682,-93.723,414.507,167.136,43.565,158.025
C01562=1028.688,-93.473,414.497,167.140,43.563,158.025
C01563=1028.694,-93.223,414.488,167.143,43.562,158.025
C01564=1028.700,-92.974,414.477,167.145,43.560,158.025
C01565=1028.706,-92.724,414.467,167.148,43.558,158.025
C01566=1028.711,-92.474,414.457,167.152,43.556,158.025
C01567=1028.717,-92.224,414.446,167.154,43.554,158.025
C01568=1028.723,-91.974,414.437,167.157,43.552,158.025
C01569=1028.729,-91.724,414.426,167.160,43.550,158.024
C01570=1028.735,-91.475,414.416,167.163,43.548,158.024
C01571=1028.741,-91.225,414.406,167.166,43.546,158.024
C01572=1028.747,-90.975,414.396,167.169,43.544,158.024
C01573=1028.752,-90.726,414.386,167.172,43.542,158.024
C01574=1028.759,-90.476,414.376,167.175,43.540,158.024
C01575=1028.764,-90.226,414.365,167.178,43.538,158.024
C01576=1028.771,-89.977,414.356,167.180,43.536,158.024
C01577=1028.776,-89.727,414.345,167.184,43.534,158.024
C01578=1028.782,-89.477,414.335,167.186,43.532,158.024
C01579=1028.788,-89.227,414.325,167.189,43.530,158.023
C01580=1028.794,-88.978,414.315,167.192,43.528,158.023
C01581=1028.800,-88.728,414.304,167.195,43.526,158.023
C01582=1028.806,-88.479,414.294,167.198,43.524,158.023
C01583=1028.812,-88.229,414.284,167.201,43.522,158.023
C01584=1028.817,-87.979,414.273,167.203,43.520,158.023
C01585=1028.824,-87.729,414.264,167.207,43.518,158.023
C01586=1028.829,-87.480,414.253,167.210,43.516,158.023
C01587=1028.836,-87.229,414.243,167.212,43.514,158.023
C01588=1028.842,-86.980,414.232,167.215,43.513,158.023
C01589=1028.848,-86.730,414.222,167.218,43.511,158.022
C01590=1028.854,-86.481,414.211,167.221,43.509,158.022
C01591=1028.860,-86.231,414.202,167.224,43.507,158.022
C01592=1028.866,-85.981,414.191,167.226,43.504,158.022
C01593=1028.871,-85.731,414.181,167.230,43.502,158.022
C01594=1028.878,-85.482,414.171,167.233,43.500,158.022
C01595=1028.883,-85.233,414.160,167.235,43.498,158.022
C01596=1028.891,-84.948,414.148,167.239,43.496,158.022
C01597=1028.898,-84.664,414.136,167.241,43.494,158.022
C01598=1028.904,-84.379,414.124,167.245,43.492,158.021
C01599=1028.911,-84.094,414.113,167.249,43.490,158.021
C01600=1028.917,-83.845,414.102,167.251,43.488,158.021
C01601=1028.923,-83.595,414.092,167.254,43.486,158.021
C01602=1028.929,-83.346,414.082,167.258,43.484,158.021
C01603=1028.936,-83.096,414.071,167.260,43.481,158.021
C01604=1028.941,-82.846,414.060,167.263,43.479,158.021
C01605=1028.948,-82.596,414.050,167.265,43.477,158.021
C01606=1028.953,-82.347,414.039,167.269,43.475,158.020
C01607=1028.960,-82.097,414.030,167.272,43.473,158.020
C01608=1028.966,-81.847,414.018,167.274,43.472,158.020
C01609=1028.972,-81.598,414.008,167.277,43.470,158.020
C01610=1028.978,-81.348,413.998,167.281,43.468,158.020
C01611=1028.984,-81.098,413.987,167.283,43.466,158.020
C01612=1028.990,-80.849,413.977,167.286,43.464,158.020
C01613=1028.996,-80.599,413.966,167.289,43.462,158.020
C01614=1029.003,-80.349,413.956,167.292,43.460,158.020
C01615=1029.008,-80.099,413.945,167.295,43.457,158.019
C01616=1029.014,-79.850,413.934,167.297,43.456,158.019
C01617=1029.020,-79.600,413.923,167.300,43.454,158.019
C01618=1029.026,-79.350,413.912,167.304,43.452,158.019
C01619=1029.032,-79.100,413.903,167.306,43.450,158.019
C01620=1029.039,-78.850,413.891,167.309,43.449,158.019
C01621=1029.044,-78.601,413.880,167.312,43.447,158.019
C01622=1029.050,-78.351,413.870,167.314,43.445,158.019
C01623=1029.056,-78.102,413.859,167.317,43.443,158.019
C01624=1029.062,-77.852,413.847,167.321,43.441,158.019
C01625=1029.069,-77.602,413.837,167.323,43.439,158.019
C01626=1029.074,-77.353,413.826,167.326,43.437,158.018
C01627=1029.080,-77.103,413.815,167.329,43.435,158.018
C01628=1029.086,-76.853,413.805,167.331,43.433,158.018
C01629=1029.092,-76.603,413.794,167.335,43.432,158.018
C01630=1029.098,-76.354,413.783,167.338,43.430,158.018
C01631=1029.104,-76.103,413.772,167.340,43.428,158.018
C01632=1029.110,-75.854,413.762,167.343,43.426,158.018
C01633=1029.116,-75.605,413.751,167.346,43.424,158.018
C01634=1029.122,-75.355,413.740,167.348,43.423,158.018
C01635=1029.128,-75.105,413.729,167.352,43.420,158.018
C01636=1029.134,-74.856,413.718,167.355,43.419,158.017
C01637=1029.140,-74.606,413.707,167.357,43.417,158.017
C01638=1029.146,-74.356,413.696,167.360,43.415,158.017
C01639=1029.152,-74.106,413.685,167.363,43.413,158.017
C01640=1029.158,-73.856,413.673,167.366,43.412,158.017
C01641=1029.164,-73.607,413.662,167.369,43.410,158.017
C01642=1029.170,-73.358,413.651,167.372,43.408,158.017
C01643=1029.176,-73.108,413.640,167.375,43.406,158.017
C01644=1029.182,-72.858,413.629,167.377,43.405,158.017
C01645=1029.188,-72.609,413.618,167.380,43.403,158.017
C01646=1029.193,-72.359,413.607,167.383,43.401,158.017
C01647=1029.199,-72.109,413.595,167.385,43.399,158.017
C01648=1029.205,-71.860,413.584,167.388,43.398,158.017
C01649=1029.212,-71.610,413.572,167.392,43.396,158.017
C01650=1029.217,-71.360,413.562,167.394,43.394,158.016
C01651=1029.223,-71.111,413.551,167.397,43.393,158.016
C01652=1029.229,-70.861,413.539,167.400,43.391,158.016
C01653=1029.235,-70.611,413.527,167.403,43.389,158.016
C01654=1029.240,-70.362,413.516,167.405,43.387,158.016
C01655=1029.247,-70.112,413.505,167.408,43.386,158.016
C01656=1029.252,-69.862,413.494,167.411,43.384,158.016
C01657=1029.259,-69.613,413.482,167.413,43.382,158.016
C01658=1029.265,-69.363,413.471,167.416,43.380,158.016
C01659=1029.270,-69.113,413.460,167.420,43.379,158.016
C01660=1029.277,-68.831,413.448,167.423,43.377,158.016
C01661=1029.284,-68.548,413.435,167.426,43.375,158.016
C01662=1029.291,-68.267,413.421,167.429,43.373,158.016
C01663=1029.297,-67.984,413.408,167.433,43.371,158.015
C01664=1029.304,-67.734,413.397,167.435,43.369,158.015
C01665=1029.309,-67.485,413.386,167.438,43.367,158.015
C01666=1029.315,-67.236,413.375,167.441,43.366,158.015
C01667=1029.322,-66.986,413.363,167.443,43.364,158.015
C01668=1029.327,-66.736,413.352,167.446,43.363,158.015
C01669=1029.333,-66.486,413.340,167.449,43.361,158.015
C01670=1029.339,-66.237,413.329,167.451,43.359,158.015
C01671=1029.346,-65.987,413.317,167.455,43.357,158.015
C01672=1029.352,-65.738,413.306,167.458,43.356,158.015
C01673=1029.357,-65.487,413.294,167.461,43.354,158.015
C01674=1029.363,-65.238,413.283,167.463,43.352,158.014
C01675=1029.369,-64.988,413.271,167.466,43.350,158.014
C01676=1029.376,-64.739,413.260,167.469,43.349,158.014
C01677=1029.382,-64.489,413.249,167.471,43.347,158.014
C01678=1029.387,-64.239,413.237,167.474,43.345,158.014
C01679=1029.394,-63.990,413.225,167.477,43.343,158.014
C01680=1029.400,-63.739,413.214,167.479,43.342,158.014
C01681=1029.406,-63.491,413.202,167.483,43.340,158.014
C01682=1029.412,-63.240,413.191,167.486,43.338,158.014
C01683=1029.418,-62.991,413.179,167.488,43.336,158.014
C01684=1029.424,-62.741,413.168,167.491,43.335,158.014
C01685=1029.430,-62.492,413.156,167.494,43.333,158.014
C01686=1029.436,-62.242,413.145,167.497,43.331,158.014
C01687=1029.443,-61.992,413.133,167.499,43.329,158.013
C01688=1029.448,-61.743,413.121,167.502,43.328,158.013
C01689=1029.455,-61.493,413.109,167.505,43.326,158.013
C01690=1029.460,-61.243,413.099,167.507,43.324,158.013
C01691=1029.467,-60.994,413.087,167.511,43.322,158.013
C01692=1029.473,-60.744,413.075,167.514,43.321,158.013
C01693=1029.479,-60.495,413.063,167.516,43.319,158.013
C01694=1029.485,-60.245,413.051,167.519,43.318,158.013
C01695=1029.491,-59.995,413.040,167.522,43.316,158.013
C01696=1029.498,-59.746,413.028,167.525,43.314,158.013
C01697=1029.503,-59.495,413.017,167.527,43.312,158.013
C01698=1029.509,-59.247,413.005,167.530,43.311,158.013
C01699=1029.516,-58.996,412.994,167.533,43.309,158.012
C01700=1029.522,-58.747,412.982,167.535,43.307,158.012
C01701=1029.528,-58.498,412.970,167.538,43.305,158.012
C01702=1029.534,-58.247,412.958,167.542,43.303,158.012
C01703=1029.541,-57.998,412.946,167.544,43.302,158.012
C01704=1029.547,-57.749,412.935,167.547,43.300,158.012
C01705=1029.552,-57.498,412.923,167.550,43.298,158.012
C01706=1029.559,-57.249,412.911,167.552,43.296,158.012
C01707=1029.566,-56.999,412.899,167.555,43.294,158.012
C01708=1029.571,-56.750,412.888,167.558,43.293,158.012
C01709=1029.577,-56.500,412.876,167.561,43.291,158.012
C01710=1029.584,-56.250,412.864,167.563,43.290,158.011
C01711=1029.590,-56.001,412.853,167.566,43.288,158.011
C01712=1029.596,-55.751,412.841,167.570,43.286,158.011
C01713=1029.602,-55.501,412.828,167.572,43.284,158.011
C01714=1029.609,-55.252,412.816,167.575,43.283,158.011
C01715=1029.614,-55.002,412.805,167.578,43.281,158.011
C01716=1029.621,-54.753,412.793,167.580,43.279,158.011
C01717=1029.627,-54.503,412.781,167.583,43.277,158.011
C01718=1029.634,-54.253,412.769,167.586,43.275,158.011
C01719=1029.639,-54.004,412.758,167.589,43.274,158.011
C01720=1029.646,-53.754,412.746,167.591,43.272,158.011
C01721=1029.652,-53.504,412.734,167.594,43.270,158.010
C01722=1029.659,-53.255,412.722,167.596,43.268,158.010
C01723=1029.665,-53.005,412.710,167.599,43.267,158.010
C01724=1029.672,-52.724,412.696,167.603,43.265,158.010
C01725=1029.679,-52.443,412.684,167.605,43.263,158.010
C01726=1029.686,-52.162,412.669,167.609,43.261,158.010
C01727=1029.693,-51.881,412.657,167.612,43.259,158.010
C01728=1029.699,-51.631,412.644,167.614,43.257,158.010
C01729=1029.705,-51.382,412.632,167.618,43.255,158.010
C01730=1029.712,-51.132,412.620,167.621,43.253,158.009
C01731=1029.719,-50.883,412.608,167.624,43.252,158.009
C01732=1029.724,-50.633,412.596,167.626,43.250,158.009
C01733=1029.731,-50.384,412.584,167.629,43.248,158.009
C01734=1029.737,-50.134,412.572,167.632,43.247,158.009
C01735=1029.742,-49.884,412.559,167.634,43.245,158.009
C01736=1029.749,-49.634,412.547,167.637,43.244,158.009
C01737=1029.755,-49.385,412.535,167.640,43.242,158.009
C01738=1029.760,-49.135,412.522,167.643,43.240,158.009
C01739=1029.767,-48.886,412.510,167.645,43.239,158.009
C01740=1029.773,-48.636,412.498,167.648,43.237,158.009
C01741=1029.779,-48.386,412.485,167.651,43.236,158.009
C01742=1029.785,-48.136,412.473,167.654,43.234,158.009
C01743=1029.791,-47.887,412.461,167.656,43.232,158.009
C01744=1029.797,-47.637,412.449,167.659,43.231,158.009
C01745=1029.803,-47.388,412.437,167.662,43.229,158.008
C01746=1029.809,-47.138,412.424,167.665,43.228,158.008
C01747=1029.815,-46.888,412.411,167.667,43.226,158.008
C01748=1029.822,-46.639,412.399,167.670,43.224,158.008
C01749=1029.828,-46.389,412.386,167.673,43.223,158.008
C01750=1029.834,-46.139,412.374,167.675,43.221,158.008
C01751=1029.841,-45.890,412.362,167.678,43.220,158.008
C01752=1029.846,-45.640,412.349,167.680,43.218,158.008
C01753=1029.852,-45.391,412.337,167.682,43.217,158.008
C01754=1029.858,-45.141,412.325,167.685,43.215,158.008
C01755=1029.865,-44.892,412.312,167.688,43.214,158.008
C01756=1029.871,-44.642,412.299,167.691,43.212,158.008
C01757=1029.877,-44.392,412.287,167.693,43.210,158.008
C01758=1029.883,-44.143,412.275,167.696,43.209,158.007
C01759=1029.889,-43.893,412.262,167.699,43.207,158.007
C01760=1029.896,-43.644,412.249,167.702,43.206,158.007
C01761=1029.902,-43.394,412.237,167.704,43.204,158.007
C01762=1029.908,-43.144,412.224,167.707,43.203,158.007
C01763=1029.914,-42.894,412.212,167.710,43.201,158.007
C01764=1029.921,-42.645,412.199,167.713,43.200,158.007
C01765=1029.927,-42.395,412.187,167.715,43.198,158.007
C01766=1029.933,-42.146,412.175,167.718,43.196,158.007
C01767=1029.939,-41.896,412.162,167.721,43.195,158.007
C01768=1029.945,-41.647,412.149,167.723,43.193,158.007
C01769=1029.951,-41.397,412.136,167.726,43.191,158.007
C01770=1029.958,-41.147,412.124,167.729,43.190,158.007
C01771=1029.964,-40.898,412.111,167.732,43.188,158.007
C01772=1029.970,-40.648,412.098,167.734,43.186,158.006
C01773=1029.977,-40.398,412.087,167.737,43.185,158.006
C01774=1029.983,-40.148,412.074,167.740,43.183,158.006
C01775=1029.989,-39.899,412.061,167.743,43.182,158.006
C01776=1029.995,-39.650,412.049,167.745,43.180,158.006
C01777=1030.002,-39.400,412.035,167.748,43.178,158.006
C01778=1030.008,-39.150,412.023,167.751,43.177,158.006
C01779=1030.013,-38.901,412.010,167.753,43.175,158.006
C01780=1030.020,-38.651,411.997,167.756,43.173,158.006
C01781=1030.026,-38.401,411.985,167.759,43.172,158.006
C01782=1030.032,-38.152,411.971,167.762,43.171,158.006
C01783=1030.038,-37.903,411.959,167.763,43.169,158.006
C01784=1030.045,-37.653,411.946,167.766,43.168,158.006
C01785=1030.051,-37.403,411.933,167.769,43.166,158.006
C01786=1030.057,-37.154,411.920,167.772,43.165,158.006
C01787=1030.063,-36.904,411.908,167.774,43.163,158.005
C01788=1030.070,-36.624,411.893,167.777,43.161,158.005
C01789=1030.076,-36.343,411.878,167.781,43.160,158.005
C01790=1030.083,-36.062,411.864,167.784,43.158,158.005
C01791=1030.090,-35.782,411.849,167.786,43.156,158.005
C01792=1030.096,-35.532,411.836,167.789,43.155,158.005
C01793=1030.102,-35.283,411.823,167.792,43.153,158.005
C01794=1030.109,-35.033,411.810,167.795,43.152,158.005
C01795=1030.114,-34.783,411.797,167.797,43.150,158.005
C01796=1030.121,-34.534,411.784,167.800,43.149,158.005
C01797=1030.127,-34.284,411.772,167.803,43.147,158.005
C01798=1030.133,-34.035,411.758,167.806,43.146,158.005
C01799=1030.140,-33.785,411.745,167.807,43.144,158.005
C01800=1030.145,-33.535,411.732,167.810,43.143,158.005
C01801=1030.152,-33.286,411.719,167.813,43.141,158.004
C01802=1030.158,-33.036,411.706,167.816,43.140,158.004
C01803=1030.164,-32.787,411.693,167.818,43.138,158.004
C01804=1030.170,-32.537,411.680,167.821,43.137,158.004
C01805=1030.176,-32.288,411.667,167.824,43.135,158.004
C01806=1030.183,-32.038,411.654,167.827,43.134,158.004
C01807=1030.190,-31.789,411.641,167.829,43.132,158.004
C01808=1030.196,-31.539,411.628,167.832,43.130,158.004
C01809=1030.202,-31.290,411.615,167.834,43.129,158.004
C01810=1030.208,-31.040,411.602,167.836,43.128,158.004
C01811=1030.214,-30.790,411.589,167.839,43.126,158.004
C01812=1030.221,-30.540,411.576,167.842,43.125,158.004
C01813=1030.227,-30.291,411.562,167.845,43.123,158.004
